  MoveL (T16343) to (117.45, 112.15, 17.7) mm, rotated rx 180 ry 0 rz -180 deg; joints [2.729, 71.249, -37.734, 4.933, -33.613, -4.112]
  Call Extruder 0.04881
  MoveL (T16344) to (118.18, 113.58, 17.7) mm, rotated rx 180 ry 0 rz -180 deg; joints [2.729, 71.249, -37.734, 4.933, -33.613, -4.112]
  Call Extruder 0.12804
  MoveL (T16345) to (121.16, 116.55, 17.7) mm, rotated rx 180 ry 0 rz -180 deg; joints [1.429, 67.441, -30.576, 2.381, -36.89, -1.905]
  Call Extruder 0.03385
  MoveL (T16346) to (121.16, 117.66, 17.7) mm, rotated rx 180 ry 0 rz -180 deg; joints [1.429, 67.441, -30.576, 2.381, -36.89, -1.905]
  Call Extruder 0.04175
  MoveL (T16347) to (120.19, 118.63, 17.7) mm, rotated rx 180 ry 0 rz -180 deg; joints [1.432, 67.145, -30.019, 2.372, -37.15, -1.891]
  Call Extruder 0.04741
  MoveL (T16348) to (120.19, 120.19, 17.7) mm, rotated rx 180 ry 0 rz -180 deg; joints [1.432, 67.145, -30.019, 2.372, -37.15, -1.891]
  Call Extruder 0.04175
  MoveL (T16349) to (121.16, 121.16, 17.7) mm, rotated rx 180 ry 0 rz -180 deg; joints [1.432, 67.145, -30.019, 2.372, -37.15, -1.891]
  Call Extruder 0.07441
  MoveL (T16350) to (121.16, 118.71, 17.7) mm, rotated rx 180 ry 0 rz -180 deg; joints [1.821, 66.26, -28.355, 2.962, -37.942, -2.336]
  Set speed (150.0 mm/s)
  MoveL (T16351) to (120.05, 117.4, 17.7) mm, rotated rx 180 ry 0 rz -180 deg; joints [1.821, 66.26, -28.355, 2.962, -37.942, -2.336]
  Set speed (50.0 mm/s)
  MoveL (T16352) to (120.05, 117.4, 17.7) mm, rotated rx 180 ry 0 rz -180 deg; joints [1.442, 66.234, -28.307, 2.345, -37.95, -1.849]
  Call Extruder 0.01089
  MoveL (T16353) to (119.96, 117.05, 17.7) mm, rotated rx 180 ry 0 rz -180 deg; joints [1.442, 66.234, -28.307, 2.345, -37.95, -1.849]
  Call Extruder 0.0635
  MoveL (T16354) to (119.01, 115.2, 17.7) mm, rotated rx 180 ry 0 rz -180 deg; joints [3.211, 71.325, -37.875, 5.812, -33.585, -4.847]
  Call Extruder 0.09231
  MoveL (T16355) to (121.16, 113.06, 17.7) mm, rotated rx 180 ry 0 rz -180 deg; joints [3.211, 71.325, -37.875, 5.812, -33.585, -4.847]
  Call Extruder 0.03385
  MoveL (T16356) to (121.16, 111.94, 17.7) mm, rotated rx 180 ry 0 rz -180 deg; joints [3.211, 71.325, -37.875, 5.812, -33.585, -4.847]
  Call Extruder 0.06789
  MoveL (T16357) to (119.58, 110.37, 17.7) mm, rotated rx 180 ry 0 rz -180 deg; joints [3.226, 70.568, -36.453, 5.738, -34.249, -4.748]
  Call Extruder 0.03053
  MoveL (T16358) to (120.29, 109.66, 17.7) mm, rotated rx 180 ry 0 rz -180 deg; joints [3.226, 70.568, -36.453, 5.738, -34.249, -4.748]
  Call Extruder 0.00661
  MoveL (T16359) to (120.37, 109.46, 17.7) mm, rotated rx 180 ry 0 rz -180 deg; joints [3.226, 70.568, -36.453, 5.738, -34.249, -4.748]
  Call Extruder 0.00686
  MoveL (T16360) to (120.37, 109.23, 17.7) mm, rotated rx 180 ry 0 rz -180 deg; joints [3.226, 70.568, -36.453, 5.738, -34.249, -4.748]
  Call Extruder 0.03378
  MoveL (T16361) to (121.16, 108.45, 17.7) mm, rotated rx 180 ry 0 rz -180 deg; joints [3.226, 70.568, -36.453, 5.738, -34.249, -4.748]
  Call Extruder 0.03385
  MoveL (T16362) to (121.16, 107.34, 17.7) mm, rotated rx 180 ry 0 rz -180 deg; joints [3.226, 70.568, -36.453, 5.738, -34.249, -4.748]
  Call Extruder 0.03378
  MoveL (T16363) to (120.37, 106.56, 17.7) mm, rotated rx 180 ry 0 rz -180 deg; joints [3.226, 70.568, -36.453, 5.738, -34.249, -4.748]
  Call Extruder 0.04531
  MoveL (T16364) to (120.37, 105.07, 17.7) mm, rotated rx 180 ry 0 rz -180 deg; joints [3.226, 70.568, -36.453, 5.738, -34.249, -4.748]
  Call Extruder 0.00661
  MoveL (T16365) to (120.29, 104.87, 17.7) mm, rotated rx 180 ry 0 rz -180 deg; joints [3.219, 70.895, -37.068, 5.77, -33.962, -4.79]
  Call Extruder 0.00334
  MoveL (T16366) to (120.21, 104.79, 17.7) mm, rotated rx 180 ry 0 rz -180 deg; joints [3.219, 70.895, -37.068, 5.77, -33.962, -4.79]
  Call Extruder 0.04071
  MoveL (T16367) to (121.16, 103.84, 17.7) mm, rotated rx 180 ry 0 rz -180 deg; joints [3.219, 70.895, -37.068, 5.77, -33.962, -4.79]
  Call Extruder 0.07441
  MoveL (T16368) to (121.16, 106.29, 17.7) mm, rotated rx 180 ry 0 rz -180 deg; joints [3.219, 70.895, -37.068, 5.77, -33.962, -4.79]
  Set speed (45.0 mm/s)
  Call Extruder -1.6
  MoveL (T16369) to (121.16, 106.29, 17.7) mm, rotated rx 180 ry 0 rz -180 deg; joints [3.219, 70.895, -37.068, 5.77, -33.962, -4.79]
  Set speed (120.0 mm/s)
  MoveL (T16370) to (121.16, 106.29, 17.7) mm, rotated rx 180 ry 0 rz -180 deg; joints [3.219, 70.895, -37.068, 5.77, -33.962, -4.79]
  Call Extruder -0.38
  MoveL (T16371) to (121.16, 105.22, 17.7) mm, rotated rx 180 ry 0 rz -180 deg; joints [3.219, 70.895, -37.068, 5.77, -33.962, -4.79]
  Set speed (45.0 mm/s)
  Call Extruder -0.02
  MoveL (T16372) to (121.16, 105.22, 17.7) mm, rotated rx 180 ry 0 rz -180 deg; joints [3.219, 70.895, -37.068, 5.77, -33.962, -4.79]
  Set speed (150.0 mm/s)
  MoveL (T16373) to (121.16, 105.22, 19.7) mm, rotated rx 180 ry 0 rz -180 deg; joints [1.407, 66.123, -28.505, 2.305, -37.64, -1.825]
  MoveL (T16374) to (120.15, 108.89, 19.7) mm, rotated rx 180 ry 0 rz -180 deg; joints [1.407, 66.336, -28.539, 2.296, -37.819, -1.814]
  MoveL (T16375) to (120.15, 108.89, 17.7) mm, rotated rx 180 ry 0 rz -180 deg; joints [1.407, 66.336, -28.539, 2.296, -37.819, -1.814]
  Set speed (40.0 mm/s)
  Call Extruder 2.0
  MoveL (T16376) to (120.15, 108.89, 17.7) mm, rotated rx 180 ry 0 rz -180 deg; joints [1.407, 66.336, -28.539, 2.296, -37.819, -1.814]
  Call Extruder 0.11511
  MoveL (T16377) to (117.48, 111.56, 17.7) mm, rotated rx 180 ry 0 rz -180 deg; joints [1.407, 66.336, -28.539, 2.296, -37.819, -1.814]
  Set speed (45.0 mm/s)
  Call Extruder -1.6
  MoveL (T16378) to (117.48, 111.56, 17.7) mm, rotated rx 180 ry 0 rz -180 deg; joints [1.407, 66.336, -28.539, 2.296, -37.819, -1.814]
  Set speed (120.0 mm/s)
  MoveL (T16379) to (117.48, 111.56, 17.7) mm, rotated rx 180 ry 0 rz -180 deg; joints [1.407, 66.336, -28.539, 2.296, -37.819, -1.814]
  Call Extruder -0.38
  MoveL (T16380) to (118.23, 110.8, 17.7) mm, rotated rx 180 ry 0 rz -180 deg; joints [1.407, 66.336, -28.539, 2.296, -37.819, -1.814]
  Set speed (45.0 mm/s)
  Call Extruder -0.02
  MoveL (T16381) to (118.23, 110.8, 17.7) mm, rotated rx 180 ry 0 rz -180 deg; joints [1.407, 66.336, -28.539, 2.296, -37.819, -1.814]
  Set speed (150.0 mm/s)
  MoveL (T16382) to (118.23, 110.8, 19.7) mm, rotated rx 180 ry 0 rz -180 deg; joints [1.407, 66.336, -28.539, 2.296, -37.819, -1.814]
  MoveL (T16383) to (118.65, 121.34, 19.7) mm, rotated rx 180 ry 0 rz -180 deg; joints [1.363, 71.176, -37.635, 2.466, -33.565, -2.055]
  MoveL (T16384) to (118.65, 121.34, 17.7) mm, rotated rx 180 ry 0 rz -180 deg; joints [1.363, 71.176, -37.635, 2.466, -33.565, -2.055]
  Set speed (40.0 mm/s)
  Call Extruder 2.0
  MoveL (T16385) to (118.65, 121.34, 17.7) mm, rotated rx 180 ry 0 rz -180 deg; joints [1.363, 71.176, -37.635, 2.466, -33.565, -2.055]
  Call Extruder 0.04796
  MoveL (T16386) to (119.76, 120.23, 17.7) mm, rotated rx 180 ry 0 rz -180 deg; joints [3.241, 71.403, -38.062, 5.883, -33.48, -4.912]
  Call Extruder 0.00166
  MoveL (T16387) to (119.78, 120.18, 17.7) mm, rotated rx 180 ry 0 rz -180 deg; joints [3.241, 71.403, -38.062, 5.883, -33.48, -4.912]
  Call Extruder 0.01669
  MoveL (T16388) to (119.78, 119.63, 17.7) mm, rotated rx 180 ry 0 rz -180 deg; joints [3.241, 71.403, -38.062, 5.883, -33.48, -4.912]
  Call Extruder 0.06581
  MoveL (T16389) to (118.25, 121.16, 17.7) mm, rotated rx 180 ry 0 rz -180 deg; joints [3.351, 66.321, -28.512, 5.456, -37.936, -4.308]
  Call Extruder 0.01758
  MoveL (T16390) to (117.68, 121.16, 17.7) mm, rotated rx 180 ry 0 rz -180 deg; joints [3.351, 66.321, -28.512, 5.456, -37.936, -4.308]
  Call Extruder 0.09068
  MoveL (T16391) to (119.78, 119.05, 17.7) mm, rotated rx 180 ry 0 rz -180 deg; joints [3.351, 66.321, -28.512, 5.456, -37.936, -4.308]
  Call Extruder 0.01758
  MoveL (T16392) to (119.78, 118.48, 17.7) mm, rotated rx 180 ry 0 rz -180 deg; joints [1.409, 66.13, -28.153, 2.29, -37.999, -1.805]
  Call Extruder 0.11554
  MoveL (T16393) to (117.1, 121.16, 17.7) mm, rotated rx 180 ry 0 rz -180 deg; joints [1.409, 66.13, -28.153, 2.29, -37.999, -1.805]
  Call Extruder 0.01758
  MoveL (T16394) to (116.52, 121.16, 17.7) mm, rotated rx 180 ry 0 rz -180 deg; joints [1.409, 66.13, -28.153, 2.29, -37.999, -1.805]
  Call Extruder 0.13957
  MoveL (T16395) to (119.76, 117.92, 17.7) mm, rotated rx 180 ry 0 rz -180 deg; joints [1.407, 66.32, -28.51, 2.295, -37.833, -1.813]
  Call Extruder 0.01457
  MoveL (T16396) to (119.65, 117.45, 17.7) mm, rotated rx 180 ry 0 rz -180 deg; joints [1.407, 66.32, -28.51, 2.295, -37.833, -1.813]
  Call Extruder 0.15961
  MoveL (T16397) to (115.95, 121.16, 17.7) mm, rotated rx 180 ry 0 rz -180 deg; joints [1.407, 66.32, -28.51, 2.295, -37.833, -1.813]
  Call Extruder 0.01758
  MoveL (T16398) to (115.37, 121.16, 17.7) mm, rotated rx 180 ry 0 rz -180 deg; joints [1.407, 66.32, -28.51, 2.295, -37.833, -1.813]
  Call Extruder 0.17783
  MoveL (T16399) to (119.49, 117.03, 17.7) mm, rotated rx 180 ry 0 rz -180 deg; joints [1.407, 66.32, -28.51, 2.295, -37.833, -1.813]
  Call Extruder 0.01306
  MoveL (T16400) to (119.3, 116.65, 17.7) mm, rotated rx 180 ry 0 rz -180 deg; joints [1.407, 66.32, -28.51, 2.295, -37.833, -1.813]
  Call Extruder 0.19428
  MoveL (T16401) to (114.8, 121.16, 17.7) mm, rotated rx 180 ry 0 rz -180 deg; joints [1.365, 66.126, -28.145, 2.218, -38.002, -1.748]
  Call Extruder 0.01758
  MoveL (T16402) to (114.22, 121.16, 17.7) mm, rotated rx 180 ry 0 rz -180 deg; joints [1.365, 66.126, -28.145, 2.218, -38.002, -1.748]
  Call Extruder 0.21073
  MoveL (T16403) to (119.1, 116.27, 17.7) mm, rotated rx 180 ry 0 rz -180 deg; joints [1.365, 66.126, -28.145, 2.218, -38.002, -1.748]
  Call Extruder 0.01306
  MoveL (T16404) to (118.91, 115.89, 17.7) mm, rotated rx 180 ry 0 rz -180 deg; joints [1.365, 66.126, -28.145, 2.218, -38.002, -1.748]
  Call Extruder 0.22717
  MoveL (T16405) to (113.64, 121.16, 17.7) mm, rotated rx 180 ry 0 rz -180 deg; joints [1.319, 71.301, -37.87, 2.394, -33.454, -1.998]
  Call Extruder 0.01758
  MoveL (T16406) to (113.07, 121.16, 17.7) mm, rotated rx 180 ry 0 rz -180 deg; joints [1.319, 71.301, -37.87, 2.394, -33.454, -1.998]
  Call Extruder 0.24362
  MoveL (T16407) to (118.71, 115.51, 17.7) mm, rotated rx 180 ry 0 rz -180 deg; joints [1.319, 71.301, -37.87, 2.394, -33.454, -1.998]
  Call Extruder 0.01306
  MoveL (T16408) to (118.52, 115.13, 17.7) mm, rotated rx 180 ry 0 rz -180 deg; joints [3.282, 71.54, -38.319, 5.974, -33.364, -4.995]
  Call Extruder 0.26007
  MoveL (T16409) to (112.49, 121.16, 17.7) mm, rotated rx 180 ry 0 rz -180 deg; joints [3.282, 71.54, -38.319, 5.974, -33.364, -4.995]
  Call Extruder 0.01758
  MoveL (T16410) to (111.91, 121.16, 17.7) mm, rotated rx 180 ry 0 rz -180 deg; joints [3.398, 66.223, -28.327, 5.521, -38.025, -4.354]
  Call Extruder 0.27651
  MoveL (T16411) to (118.32, 114.75, 17.7) mm, rotated rx 180 ry 0 rz -180 deg; joints [3.398, 66.223, -28.327, 5.521, -38.025, -4.354]
  Call Extruder 0.01306
  MoveL (T16412) to (118.13, 114.36, 17.7) mm, rotated rx 180 ry 0 rz -180 deg; joints [3.398, 66.223, -28.327, 5.521, -38.025, -4.354]
  Call Extruder 0.29296
  MoveL (T16413) to (111.34, 121.16, 17.7) mm, rotated rx 180 ry 0 rz -180 deg; joints [3.398, 66.223, -28.327, 5.521, -38.025, -4.354]
  Call Extruder 0.01758
  MoveL (T16414) to (110.76, 121.16, 17.7) mm, rotated rx 180 ry 0 rz -180 deg; joints [1.366, 66.024, -27.953, 2.215, -38.092, -1.744]
  Call Extruder 0.30941
  MoveL (T16415) to (117.93, 113.98, 17.7) mm, rotated rx 180 ry 0 rz -180 deg; joints [1.366, 66.024, -27.953, 2.215, -38.092, -1.744]
  Call Extruder 0.01306
  MoveL (T16416) to (117.74, 113.6, 17.7) mm, rotated rx 180 ry 0 rz -180 deg; joints [1.366, 66.024, -27.953, 2.215, -38.092, -1.744]
  Call Extruder 0.32585
  MoveL (T16417) to (110.18, 121.16, 17.7) mm, rotated rx 180 ry 0 rz -180 deg; joints [1.365, 66.111, -28.116, 2.217, -38.015, -1.747]
  Call Extruder 0.01758
  MoveL (T16418) to (109.61, 121.16, 17.7) mm, rotated rx 180 ry 0 rz -180 deg; joints [1.365, 66.111, -28.116, 2.217, -38.015, -1.747]
  Call Extruder 0.3423
  MoveL (T16419) to (117.54, 113.22, 17.7) mm, rotated rx 180 ry 0 rz -180 deg; joints [1.365, 66.111, -28.116, 2.217, -38.015, -1.747]
  Call Extruder 0.01306
  MoveL (T16420) to (117.35, 112.84, 17.7) mm, rotated rx 180 ry 0 rz -180 deg; joints [1.365, 66.111, -28.116, 2.217, -38.015, -1.747]
  Call Extruder 0.35875
  MoveL (T16421) to (109.03, 121.16, 17.7) mm, rotated rx 180 ry 0 rz -180 deg; joints [1.332, 65.919, -27.755, 2.156, -38.183, -1.695]
  Call Extruder 0.01758
  MoveL (T16422) to (108.45, 121.16, 17.7) mm, rotated rx 180 ry 0 rz -180 deg; joints [1.332, 65.919, -27.755, 2.156, -38.183, -1.695]
  Call Extruder 0.37519
  MoveL (T16423) to (117.15, 112.46, 17.7) mm, rotated rx 180 ry 0 rz -180 deg; joints [1.332, 65.919, -27.755, 2.156, -38.183, -1.695]
  Call Extruder 0.01306
  MoveL (T16424) to (116.96, 112.08, 17.7) mm, rotated rx 180 ry 0 rz -180 deg; joints [1.332, 65.919, -27.755, 2.156, -38.183, -1.695]
  Call Extruder 0.39164
  MoveL (T16425) to (107.88, 121.16, 17.7) mm, rotated rx 180 ry 0 rz -180 deg; joints [1.332, 65.919, -27.755, 2.156, -38.183, -1.695]
  Call Extruder 0.01758
  MoveL (T16426) to (107.3, 121.16, 17.7) mm, rotated rx 180 ry 0 rz -180 deg; joints [1.332, 65.919, -27.755, 2.156, -38.183, -1.695]
  Call Extruder 0.40809
  MoveL (T16427) to (116.76, 111.69, 17.7) mm, rotated rx 180 ry 0 rz -180 deg; joints [1.332, 65.919, -27.755, 2.156, -38.183, -1.695]
  Call Extruder 0.01107
  MoveL (T16428) to (116.6, 111.37, 17.7) mm, rotated rx 180 ry 0 rz -180 deg; joints [1.323, 65.918, -27.754, 2.141, -38.183, -1.683]
  Call Extruder 0.0149
  MoveL (T16429) to (117.09, 111.37, 17.7) mm, rotated rx 180 ry 0 rz -180 deg; joints [1.323, 65.918, -27.754, 2.141, -38.183, -1.683]
  Call Extruder 0.12417
  MoveL (T16430) to (119.96, 108.49, 17.7) mm, rotated rx 180 ry 0 rz -180 deg; joints [1.323, 65.918, -27.754, 2.141, -38.183, -1.683]
  Call Extruder 0.01758
  MoveL (T16431) to (119.96, 107.92, 17.7) mm, rotated rx 180 ry 0 rz -180 deg; joints [1.276, 71.427, -38.107, 2.322, -33.342, -1.94]
  Call Extruder 0.57106
  MoveL (T16432) to (106.73, 121.16, 17.7) mm, rotated rx 180 ry 0 rz -180 deg; joints [1.276, 71.427, -38.107, 2.322, -33.342, -1.94]
  Call Extruder 0.00679
  MoveL (T16433) to (106.5, 121.16, 17.7) mm, rotated rx 180 ry 0 rz -180 deg; joints [1.276, 71.427, -38.107, 2.322, -33.342, -1.94]
  Call Extruder 0.00763
  MoveL (T16434) to (106.33, 120.98, 17.7) mm, rotated rx 180 ry 0 rz -180 deg; joints [1.276, 71.427, -38.107, 2.322, -33.342, -1.94]
  Call Extruder 0.58829
  MoveL (T16435) to (119.96, 107.34, 17.7) mm, rotated rx 180 ry 0 rz -180 deg; joints [3.322, 71.677, -38.577, 6.066, -33.247, -5.079]
  Call Extruder 0.01758
  MoveL (T16436) to (119.96, 106.76, 17.7) mm, rotated rx 180 ry 0 rz -180 deg; joints [3.322, 71.677, -38.577, 6.066, -33.247, -5.079]
  Call Extruder 0.60072
  MoveL (T16437) to (106.04, 120.69, 17.7) mm, rotated rx 180 ry 0 rz -180 deg; joints [3.322, 71.677, -38.577, 6.066, -33.247, -5.079]
  Call Extruder 0.01243
  MoveL (T16438) to (105.75, 120.4, 17.7) mm, rotated rx 180 ry 0 rz -180 deg; joints [3.445, 66.125, -28.143, 5.586, -38.114, -4.4]
  Call Extruder 0.61315
  MoveL (T16439) to (119.96, 106.19, 17.7) mm, rotated rx 180 ry 0 rz -180 deg; joints [3.445, 66.125, -28.143, 5.586, -38.114, -4.4]
  Call Extruder 0.01758
  MoveL (T16440) to (119.96, 105.61, 17.7) mm, rotated rx 180 ry 0 rz -180 deg; joints [3.445, 66.125, -28.143, 5.586, -38.114, -4.4]
  Call Extruder 0.62159
  MoveL (T16441) to (105.55, 120.02, 17.7) mm, rotated rx 180 ry 0 rz -180 deg; joints [3.445, 66.125, -28.143, 5.586, -38.114, -4.4]
  Call Extruder 0.01758
  MoveL (T16442) to (105.55, 119.44, 17.7) mm, rotated rx 180 ry 0 rz -180 deg; joints [1.339, 65.919, -27.756, 2.166, -38.183, -1.703]
  Call Extruder 0.61978
  MoveL (T16443) to (119.92, 105.08, 17.7) mm, rotated rx 180 ry 0 rz -180 deg; joints [1.339, 65.919, -27.756, 2.166, -38.183, -1.703]
  Call Extruder 0.01243
  MoveL (T16444) to (119.63, 104.79, 17.7) mm, rotated rx 180 ry 0 rz -180 deg; joints [1.326, 65.933, -27.783, 2.146, -38.17, -1.687]
  Call Extruder 0.60735
  MoveL (T16445) to (105.55, 118.87, 17.7) mm, rotated rx 180 ry 0 rz -180 deg; joints [1.326, 65.933, -27.783, 2.146, -38.17, -1.687]
  Call Extruder 0.01758
  MoveL (T16446) to (105.55, 118.29, 17.7) mm, rotated rx 180 ry 0 rz -180 deg; joints [1.326, 65.933, -27.783, 2.146, -38.17, -1.687]
  Call Extruder 0.59492
  MoveL (T16447) to (119.35, 104.5, 17.7) mm, rotated rx 180 ry 0 rz -180 deg; joints [1.326, 65.933, -27.783, 2.146, -38.17, -1.687]
  Call Extruder 0.01243
  MoveL (T16448) to (119.06, 104.21, 17.7) mm, rotated rx 180 ry 0 rz -180 deg; joints [1.326, 65.933, -27.783, 2.146, -38.17, -1.687]
  Call Extruder 0.58249
  MoveL (T16449) to (105.55, 117.72, 17.7) mm, rotated rx 180 ry 0 rz -180 deg; joints [1.326, 65.933, -27.783, 2.146, -38.17, -1.687]
  Call Extruder 0.01758
  MoveL (T16450) to (105.55, 117.14, 17.7) mm, rotated rx 180 ry 0 rz -180 deg; joints [1.326, 65.933, -27.783, 2.146, -38.17, -1.687]
  Call Extruder 0.57006
  MoveL (T16451) to (118.77, 103.92, 17.7) mm, rotated rx 180 ry 0 rz -180 deg; joints [1.326, 65.933, -27.783, 2.146, -38.17, -1.687]
  Call Extruder 0.00343
  MoveL (T16452) to (118.69, 103.84, 17.7) mm, rotated rx 180 ry 0 rz -180 deg; joints [1.323, 65.918, -27.754, 2.141, -38.183, -1.683]
  Call Extruder 0.01274
  MoveL (T16453) to (118.27, 103.84, 17.7) mm, rotated rx 180 ry 0 rz -180 deg; joints [1.323, 65.918, -27.754, 2.141, -38.183, -1.683]
  Call Extruder 0.54862
  MoveL (T16454) to (105.55, 116.56, 17.7) mm, rotated rx 180 ry 0 rz -180 deg; joints [1.321, 66.153, -28.196, 2.147, -37.977, -1.693]
  Call Extruder 0.01758
  MoveL (T16455) to (105.55, 115.99, 17.7) mm, rotated rx 180 ry 0 rz -180 deg; joints [1.321, 66.153, -28.196, 2.147, -37.977, -1.693]
  Call Extruder 0.0956
  MoveL (T16456) to (107.77, 113.77, 17.7) mm, rotated rx 180 ry 0 rz -180 deg; joints [1.321, 66.153, -28.196, 2.147, -37.977, -1.693]
  Set speed (150.0 mm/s)
  MoveL (T16457) to (108.15, 113.39, 17.7) mm, rotated rx 180 ry 0 rz -180 deg; joints [1.321, 66.153, -28.196, 2.147, -37.977, -1.693]
  Set speed (40.0 mm/s)
  MoveL (T16458) to (108.15, 113.39, 17.7) mm, rotated rx 180 ry 0 rz -180 deg; joints [1.321, 66.153, -28.196, 2.147, -37.977, -1.693]
  Call Extruder 0.41176
  MoveL (T16459) to (117.7, 103.84, 17.7) mm, rotated rx 180 ry 0 rz -180 deg; joints [1.321, 66.153, -28.196, 2.147, -37.977, -1.693]
  Call Extruder 0.01758
  MoveL (T16460) to (117.12, 103.84, 17.7) mm, rotated rx 180 ry 0 rz -180 deg; joints [1.321, 66.153, -28.196, 2.147, -37.977, -1.693]
  Call Extruder 0.38942
  MoveL (T16461) to (108.09, 112.87, 17.7) mm, rotated rx 180 ry 0 rz -180 deg; joints [1.321, 66.153, -28.196, 2.147, -37.977, -1.693]
  Call Extruder 0.01307
  MoveL (T16462) to (107.9, 112.49, 17.7) mm, rotated rx 180 ry 0 rz -180 deg; joints [1.321, 65.916, -28.158, 2.157, -37.777, -1.705]
  Call Extruder 0.37296
  MoveL (T16463) to (116.54, 103.84, 17.7) mm, rotated rx 180 ry 0 rz -180 deg; joints [1.402, 70.099, -36.007, 2.501, -34.117, -2.071]
  Call Extruder 0.01758
  MoveL (T16464) to (115.97, 103.84, 17.7) mm, rotated rx 180 ry 0 rz -180 deg; joints [1.402, 70.099, -36.007, 2.501, -34.117, -2.071]
  Call Extruder 0.35649
  MoveL (T16465) to (107.7, 112.11, 17.7) mm, rotated rx 180 ry 0 rz -180 deg; joints [1.402, 70.332, -36.05, 2.488, -34.308, -2.056]
  Call Extruder 0.01307
  MoveL (T16466) to (107.51, 111.73, 17.7) mm, rotated rx 180 ry 0 rz -180 deg; joints [1.402, 70.332, -36.05, 2.488, -34.308, -2.056]
  Call Extruder 0.34003
  MoveL (T16467) to (115.39, 103.84, 17.7) mm, rotated rx 180 ry 0 rz -180 deg; joints [1.402, 70.332, -36.05, 2.488, -34.308, -2.056]
  Call Extruder 0.01758
  MoveL (T16468) to (114.81, 103.84, 17.7) mm, rotated rx 180 ry 0 rz -180 deg; joints [1.402, 70.332, -36.05, 2.488, -34.308, -2.056]
  Call Extruder 0.32357
  MoveL (T16469) to (107.31, 111.35, 17.7) mm, rotated rx 180 ry 0 rz -180 deg; joints [1.402, 70.332, -36.05, 2.488, -34.308, -2.056]
  Call Extruder 0.01307
  MoveL (T16470) to (107.12, 110.96, 17.7) mm, rotated rx 180 ry 0 rz -180 deg; joints [1.402, 70.332, -36.05, 2.488, -34.308, -2.056]
  Call Extruder 0.3071
  MoveL (T16471) to (114.24, 103.84, 17.7) mm, rotated rx 180 ry 0 rz -180 deg; joints [1.402, 70.332, -36.05, 2.488, -34.308, -2.056]
  Call Extruder 0.01758
  MoveL (T16472) to (113.66, 103.84, 17.7) mm, rotated rx 180 ry 0 rz -180 deg; joints [1.396, 71.083, -37.46, 2.52, -33.648, -2.098]
  Call Extruder 0.29064
  MoveL (T16473) to (106.92, 110.58, 17.7) mm, rotated rx 180 ry 0 rz -180 deg; joints [1.396, 71.083, -37.46, 2.52, -33.648, -2.098]
  Call Extruder 0.01307
  MoveL (T16474) to (106.73, 110.2, 17.7) mm, rotated rx 180 ry 0 rz -180 deg; joints [1.396, 71.083, -37.46, 2.52, -33.648, -2.098]
  Call Extruder 0.27417
  MoveL (T16475) to (113.08, 103.84, 17.7) mm, rotated rx 180 ry 0 rz -180 deg; joints [3.316, 66.395, -28.651, 5.407, -37.868, -4.274]
  Call Extruder 0.01758
  MoveL (T16476) to (112.51, 103.84, 17.7) mm, rotated rx 180 ry 0 rz -180 deg; joints [3.316, 66.395, -28.651, 5.407, -37.868, -4.274]
  Call Extruder 0.25771
  MoveL (T16477) to (106.53, 109.82, 17.7) mm, rotated rx 180 ry 0 rz -180 deg; joints [3.316, 66.395, -28.651, 5.407, -37.868, -4.274]
  Call Extruder 0.01307
  MoveL (T16478) to (106.34, 109.44, 17.7) mm, rotated rx 180 ry 0 rz -180 deg; joints [2.938, 66.346, -28.558, 4.788, -37.885, -3.782]
  Call Extruder 0.24124
  MoveL (T16479) to (111.93, 103.84, 17.7) mm, rotated rx 180 ry 0 rz -180 deg; joints [2.938, 66.346, -28.558, 4.788, -37.885, -3.782]
  Call Extruder 0.01758
  MoveL (T16480) to (111.36, 103.84, 17.7) mm, rotated rx 180 ry 0 rz -180 deg; joints [2.938, 66.346, -28.558, 4.788, -37.885, -3.782]
  Call Extruder 0.22478
  MoveL (T16481) to (106.14, 109.06, 17.7) mm, rotated rx 180 ry 0 rz -180 deg; joints [2.938, 66.346, -28.558, 4.788, -37.885, -3.782]
  Call Extruder 0.01307
  MoveL (T16482) to (105.95, 108.67, 17.7) mm, rotated rx 180 ry 0 rz -180 deg; joints [2.938, 66.346, -28.558, 4.788, -37.885, -3.782]
  Call Extruder 0.20831
  MoveL (T16483) to (110.78, 103.84, 17.7) mm, rotated rx 180 ry 0 rz -180 deg; joints [3.295, 67.312, -30.372, 5.471, -37.065, -4.371]
  Call Extruder 0.01758
  MoveL (T16484) to (110.2, 103.84, 17.7) mm, rotated rx 180 ry 0 rz -180 deg; joints [3.295, 67.312, -30.372, 5.471, -37.065, -4.371]
  Call Extruder 0.19185
  MoveL (T16485) to (105.75, 108.29, 17.7) mm, rotated rx 180 ry 0 rz -180 deg; joints [3.295, 67.312, -30.372, 5.471, -37.065, -4.371]
  Call Extruder 0.00693
  MoveL (T16486) to (105.65, 108.09, 17.7) mm, rotated rx 180 ry 0 rz -180 deg; joints [3.288, 67.61, -30.932, 5.493, -36.804, -4.403]
  Call Extruder 0.00686
  MoveL (T16487) to (105.6, 107.87, 17.7) mm, rotated rx 180 ry 0 rz -180 deg; joints [3.288, 67.61, -30.932, 5.493, -36.804, -4.403]
  Call Extruder 0.17364
  MoveL (T16488) to (109.63, 103.84, 17.7) mm, rotated rx 180 ry 0 rz -180 deg; joints [1.879, 71.124, -37.537, 3.395, -33.633, -2.827]
  Call Extruder 0.01758
  MoveL (T16489) to (109.05, 103.84, 17.7) mm, rotated rx 180 ry 0 rz -180 deg; joints [1.879, 71.124, -37.537, 3.395, -33.633, -2.827]
  Call Extruder 0.15359
  MoveL (T16490) to (105.49, 107.41, 17.7) mm, rotated rx 180 ry 0 rz -180 deg; joints [1.879, 71.124, -37.537, 3.395, -33.633, -2.827]
  Call Extruder 0.00278
  MoveL (T16491) to (105.47, 107.32, 17.7) mm, rotated rx 180 ry 0 rz -180 deg; joints [1.879, 71.124, -37.537, 3.395, -33.633, -2.827]
  Call Extruder 0.01427
  MoveL (T16492) to (105.47, 106.85, 17.7) mm, rotated rx 180 ry 0 rz -180 deg; joints [1.879, 71.124, -37.537, 3.395, -33.633, -2.827]
  Call Extruder 0.12957
  MoveL (T16493) to (108.47, 103.84, 17.7) mm, rotated rx 180 ry 0 rz -180 deg; joints [1.763, 71.113, -37.517, 3.183, -33.637, -2.651]
  Call Extruder 0.01758
  MoveL (T16494) to (107.9, 103.84, 17.7) mm, rotated rx 180 ry 0 rz -180 deg; joints [1.763, 71.113, -37.517, 3.183, -33.637, -2.651]
  Call Extruder 0.1047
  MoveL (T16495) to (105.47, 106.27, 17.7) mm, rotated rx 180 ry 0 rz -180 deg; joints [1.763, 71.113, -37.517, 3.183, -33.637, -2.651]
  Call Extruder 0.01758
  MoveL (T16496) to (105.47, 105.69, 17.7) mm, rotated rx 180 ry 0 rz -180 deg; joints [1.405, 70.017, -35.456, 2.476, -34.585, -2.039]
  Call Extruder 0.07984
  MoveL (T16497) to (107.32, 103.84, 17.7) mm, rotated rx 180 ry 0 rz -180 deg; joints [1.405, 70.017, -35.456, 2.476, -34.585, -2.039]
  Call Extruder 0.01758
  MoveL (T16498) to (106.75, 103.84, 17.7) mm, rotated rx 180 ry 0 rz -180 deg; joints [1.408, 69.688, -34.839, 2.463, -34.874, -2.021]
  Call Extruder 0.06288
  MoveL (T16499) to (105.29, 105.3, 17.7) mm, rotated rx 180 ry 0 rz -180 deg; joints [1.408, 69.688, -34.839, 2.463, -34.874, -2.021]
  Set speed (45.0 mm/s)
  Call Extruder -1.6
  MoveL (T16500) to (105.29, 105.3, 17.7) mm, rotated rx 180 ry 0 rz -180 deg; joints [2.818, 66.332, -28.531, 4.592, -37.89, -3.627]
  Set speed (120.0 mm/s)
  MoveL (T16501) to (105.29, 105.3, 17.7) mm, rotated rx 180 ry 0 rz -180 deg; joints [2.44, 66.29, -28.454, 3.973, -37.903, -3.137]
  Call Extruder -0.38
  MoveL (T16502) to (106.04, 104.55, 17.7) mm, rotated rx 180 ry 0 rz -180 deg; joints [2.44, 66.29, -28.454, 3.973, -37.903, -3.137]
  Set speed (45.0 mm/s)
  Call Extruder -0.02
  MoveL (T16503) to (106.04, 104.55, 17.7) mm, rotated rx 180 ry 0 rz -180 deg; joints [2.44, 66.29, -28.454, 3.973, -37.903, -3.137]
  Set speed (150.0 mm/s)
  MoveL (T16504) to (106.04, 104.55, 19.7) mm, rotated rx 180 ry 0 rz -180 deg; joints [3.266, 68.57, -32.736, 5.568, -35.962, -4.511]
  MoveL (T16505) to (104.34, 103.54, 19.7) mm, rotated rx 180 ry 0 rz -180 deg; joints [3.266, 68.57, -32.736, 5.568, -35.962, -4.511]
  MoveL (T16506) to (104.34, 103.54, 17.9) mm, rotated rx 180 ry 0 rz -180 deg; joints [3.266, 68.57, -32.736, 5.568, -35.962, -4.511]
  Set speed (40.0 mm/s)
  Call Extruder 2.0
  MoveL (T16507) to (104.34, 103.54, 17.9) mm, rotated rx 180 ry 0 rz -180 deg; joints [3.266, 68.57, -32.736, 5.568, -35.962, -4.511]
  Call Extruder 0.52159
  MoveL (T16508) to (121.46, 103.54, 17.9) mm, rotated rx 180 ry 0 rz -180 deg; joints [3.26, 68.883, -33.326, 5.593, -35.687, -4.548]
  Call Extruder 0.54596
  MoveL (T16509) to (121.46, 121.46, 17.9) mm, rotated rx 180 ry 0 rz -180 deg; joints [3.26, 68.883, -33.326, 5.593, -35.687, -4.548]
  Call Extruder 0.54596
  MoveL (T16510) to (103.54, 121.46, 17.9) mm, rotated rx 180 ry 0 rz -180 deg; joints [3.26, 68.883, -33.326, 5.593, -35.687, -4.548]
  Call Extruder 0.54596
  MoveL (T16511) to (103.54, 103.54, 17.9) mm, rotated rx 180 ry 0 rz -180 deg; joints [3.26, 68.883, -33.326, 5.593, -35.687, -4.548]
  Call Extruder 0.02254
  MoveL (T16512) to (104.28, 103.54, 17.9) mm, rotated rx 180 ry 0 rz -180 deg; joints [2.362, 71.177, -37.638, 4.27, -33.613, -3.558]
  Set speed (150.0 mm/s)
  MoveL (T16513) to (103.53, 103.13, 17.9) mm, rotated rx 180 ry 0 rz -180 deg; joints [2.362, 71.177, -37.638, 4.27, -33.613, -3.558]
  Set speed (40.0 mm/s)
  MoveL (T16514) to (103.53, 103.13, 17.9) mm, rotated rx 180 ry 0 rz -180 deg; joints [2.362, 71.177, -37.638, 4.27, -33.613, -3.558]
  Call Extruder 0.55858
  MoveL (T16515) to (121.87, 103.13, 17.9) mm, rotated rx 180 ry 0 rz -180 deg; joints [2.362, 71.177, -37.638, 4.27, -33.613, -3.558]
  Call Extruder 0.57077
  MoveL (T16516) to (121.87, 121.87, 17.9) mm, rotated rx 180 ry 0 rz -180 deg; joints [2.246, 71.163, -37.611, 4.059, -33.618, -3.382]
  Call Extruder 0.57077
  MoveL (T16517) to (103.13, 121.87, 17.9) mm, rotated rx 180 ry 0 rz -180 deg; joints [2.246, 71.163, -37.611, 4.059, -33.618, -3.382]
  Call Extruder 0.57077
  MoveL (T16518) to (103.13, 103.13, 17.9) mm, rotated rx 180 ry 0 rz -180 deg; joints [2.246, 71.163, -37.611, 4.059, -33.618, -3.382]
  Call Extruder 0.01036
  MoveL (T16519) to (103.47, 103.13, 17.9) mm, rotated rx 180 ry 0 rz -180 deg; joints [1.417, 68.683, -32.95, 2.425, -35.758, -1.969]
  Set speed (150.0 mm/s)
  MoveL (T16520) to (102.72, 102.81, 17.9) mm, rotated rx 180 ry 0 rz -180 deg; joints [1.417, 68.683, -32.95, 2.425, -35.758, -1.969]
  Set speed (25.0 mm/s)
  MoveL (T16521) to (102.72, 102.81, 17.9) mm, rotated rx 180 ry 0 rz -180 deg; joints [1.42, 68.372, -32.365, 2.414, -36.032, -1.953]
  Call Extruder 0.00259
  MoveL (T16522) to (102.72, 102.72, 17.9) mm, rotated rx 180 ry 0 rz -180 deg; joints [1.42, 68.372, -32.365, 2.414, -36.032, -1.953]
  Call Extruder 0.59557
  MoveL (T16523) to (122.28, 102.72, 17.9) mm, rotated rx 180 ry 0 rz -180 deg; joints [1.42, 68.372, -32.365, 2.414, -36.032, -1.953]
  Call Extruder 0.59557
  MoveL (T16524) to (122.28, 122.28, 17.9) mm, rotated rx 180 ry 0 rz -180 deg; joints [1.42, 68.372, -32.365, 2.414, -36.032, -1.953]
  Call Extruder 0.59557
  MoveL (T16525) to (102.72, 122.28, 17.9) mm, rotated rx 180 ry 0 rz -180 deg; joints [2.319, 66.279, -28.432, 3.777, -37.907, -2.982]
  Call Extruder 0.59115
  MoveL (T16526) to (102.72, 102.87, 17.9) mm, rotated rx 180 ry 0 rz -180 deg; joints [2.319, 66.279, -28.432, 3.777, -37.907, -2.982]
  Set speed (150.0 mm/s)
  MoveL (T16527) to (102.78, 102.75, 17.9) mm, rotated rx 180 ry 0 rz -180 deg; joints [1.941, 66.245, -28.369, 3.159, -37.919, -2.493]
  Set speed (45.0 mm/s)
  Call Extruder -1.6
  MoveL (T16528) to (102.78, 102.75, 17.9) mm, rotated rx 180 ry 0 rz -180 deg; joints [1.941, 66.245, -28.369, 3.159, -37.919, -2.493]
  Set speed (120.0 mm/s)
  MoveL (T16529) to (102.78, 102.75, 17.9) mm, rotated rx 180 ry 0 rz -180 deg; joints [3.239, 69.895, -35.228, 5.681, -34.799, -4.67]
  Call Extruder -0.05166
  MoveL (T16530) to (102.72, 102.72, 17.9) mm, rotated rx 180 ry 0 rz -180 deg; joints [3.239, 69.895, -35.228, 5.681, -34.799, -4.67]
  Call Extruder -0.32834
  MoveL (T16531) to (103.65, 102.72, 17.9) mm, rotated rx 180 ry 0 rz -180 deg; joints [3.239, 69.895, -35.228, 5.681, -34.799, -4.67]
  Set speed (45.0 mm/s)
  Call Extruder -0.02
  MoveL (T16532) to (103.65, 102.72, 17.9) mm, rotated rx 180 ry 0 rz -180 deg; joints [3.232, 70.227, -35.851, 5.711, -34.509, -4.711]
  Set speed (150.0 mm/s)
  MoveL (T16533) to (103.65, 102.72, 19.9) mm, rotated rx 180 ry 0 rz -180 deg; joints [2.845, 71.243, -37.761, 5.148, -33.588, -4.292]
  MoveL (T16534) to (106.08, 103.93, 19.9) mm, rotated rx 180 ry 0 rz -180 deg; joints [2.845, 71.243, -37.761, 5.148, -33.588, -4.292]
  MoveL (T16535) to (106.08, 103.93, 17.9) mm, rotated rx 180 ry 0 rz -180 deg; joints [2.845, 71.243, -37.761, 5.148, -33.588, -4.292]
  Set speed (40.0 mm/s)
  Call Extruder 2.0
  MoveL (T16536) to (106.08, 103.93, 17.9) mm, rotated rx 180 ry 0 rz -180 deg; joints [2.845, 71.243, -37.761, 5.148, -33.588, -4.292]
  Set speed (50.0 mm/s)
  MoveL (T16537) to (106.08, 103.93, 17.9) mm, rotated rx 180 ry 0 rz -180 deg; joints [2.729, 71.226, -37.729, 4.936, -33.595, -4.115]
  Call Extruder 0.00361
  MoveL (T16538) to (106.17, 103.84, 17.9) mm, rotated rx 180 ry 0 rz -180 deg; joints [2.729, 71.226, -37.729, 4.936, -33.595, -4.115]
  Call Extruder 0.0708
  MoveL (T16539) to (103.84, 103.84, 17.9) mm, rotated rx 180 ry 0 rz -180 deg; joints [2.729, 71.226, -37.729, 4.936, -33.595, -4.115]
  Call Extruder 0.05255
  MoveL (T16540) to (105.06, 105.06, 17.9) mm, rotated rx 180 ry 0 rz -180 deg; joints [2.729, 71.226, -37.729, 4.936, -33.595, -4.115]
  Call Extruder 0.03217
  MoveL (T16541) to (105.06, 106.12, 17.9) mm, rotated rx 180 ry 0 rz -180 deg; joints [1.429, 67.418, -30.572, 2.382, -36.87, -1.906]
  Call Extruder 0.0525
  MoveL (T16542) to (103.84, 107.34, 17.9) mm, rotated rx 180 ry 0 rz -180 deg; joints [1.429, 67.418, -30.572, 2.382, -36.87, -1.906]
  Call Extruder 0.03385
  MoveL (T16543) to (103.84, 108.45, 17.9) mm, rotated rx 180 ry 0 rz -180 deg; joints [1.432, 67.122, -30.015, 2.373, -37.13, -1.892]
  Call Extruder 0.13495
  MoveL (T16544) to (106.98, 111.58, 17.9) mm, rotated rx 180 ry 0 rz -180 deg; joints [1.432, 67.122, -30.015, 2.373, -37.13, -1.892]
  Call Extruder 0.04156
  MoveL (T16545) to (107.6, 112.8, 17.9) mm, rotated rx 180 ry 0 rz -180 deg; joints [1.432, 67.122, -30.015, 2.373, -37.13, -1.892]
  Call Extruder 0.16166
  MoveL (T16546) to (103.84, 116.55, 17.9) mm, rotated rx 180 ry 0 rz -180 deg; joints [1.821, 66.236, -28.351, 2.963, -37.922, -2.338]
  Call Extruder 0.03385
  MoveL (T16547) to (103.84, 117.66, 17.9) mm, rotated rx 180 ry 0 rz -180 deg; joints [1.821, 66.236, -28.351, 2.963, -37.922, -2.338]
  Call Extruder 0.05612
  MoveL (T16548) to (105.15, 118.96, 17.9) mm, rotated rx 180 ry 0 rz -180 deg; joints [1.821, 66.236, -28.351, 2.963, -37.922, -2.338]
  Call Extruder 0.02709
  MoveL (T16549) to (105.15, 119.85, 17.9) mm, rotated rx 180 ry 0 rz -180 deg; joints [1.821, 66.236, -28.351, 2.963, -37.922, -2.338]
  Call Extruder 0.05612
  MoveL (T16550) to (103.84, 121.16, 17.9) mm, rotated rx 180 ry 0 rz -180 deg; joints [1.442, 66.21, -28.303, 2.346, -37.93, -1.851]
  Call Extruder 0.06345
  MoveL (T16551) to (105.93, 121.16, 17.9) mm, rotated rx 180 ry 0 rz -180 deg; joints [1.442, 66.21, -28.303, 2.346, -37.93, -1.851]
  Call Extruder 0.01096
  MoveL (T16552) to (105.67, 120.9, 17.9) mm, rotated rx 180 ry 0 rz -180 deg; joints [1.442, 66.21, -28.303, 2.346, -37.93, -1.851]
  Set speed (45.0 mm/s)
  Call Extruder -1.6
  MoveL (T16553) to (105.67, 120.9, 17.9) mm, rotated rx 180 ry 0 rz -180 deg; joints [3.211, 71.301, -37.871, 5.815, -33.566, -4.85]
  Set speed (120.0 mm/s)
  MoveL (T16554) to (105.67, 120.9, 17.9) mm, rotated rx 180 ry 0 rz -180 deg; joints [3.211, 71.301, -37.871, 5.815, -33.566, -4.85]
  Call Extruder -0.12811
  MoveL (T16555) to (105.93, 121.16, 17.9) mm, rotated rx 180 ry 0 rz -180 deg; joints [3.226, 70.545, -36.448, 5.741, -34.23, -4.752]
  Call Extruder -0.25189
  MoveL (T16556) to (105.22, 121.16, 17.9) mm, rotated rx 180 ry 0 rz -180 deg; joints [3.226, 70.545, -36.448, 5.741, -34.23, -4.752]
  Set speed (45.0 mm/s)
  Call Extruder -0.02
  MoveL (T16557) to (105.22, 121.16, 17.9) mm, rotated rx 180 ry 0 rz -180 deg; joints [3.226, 70.545, -36.448, 5.741, -34.23, -4.752]
  Set speed (150.0 mm/s)
  MoveL (T16558) to (105.22, 121.16, 19.9) mm, rotated rx 180 ry 0 rz -180 deg; joints [3.226, 70.545, -36.448, 5.741, -34.23, -4.752]
  MoveL (T16559) to (105.15, 117.23, 19.9) mm, rotated rx 180 ry 0 rz -180 deg; joints [3.226, 70.545, -36.448, 5.741, -34.23, -4.752]
  MoveL (T16560) to (105.15, 117.23, 17.9) mm, rotated rx 180 ry 0 rz -180 deg; joints [3.226, 70.545, -36.448, 5.741, -34.23, -4.752]
  Set speed (40.0 mm/s)
  Call Extruder 2.0
  MoveL (T16561) to (105.15, 117.23, 17.9) mm, rotated rx 180 ry 0 rz -180 deg; joints [3.226, 70.545, -36.448, 5.741, -34.23, -4.752]
  Set speed (50.0 mm/s)
  MoveL (T16562) to (105.15, 117.23, 17.9) mm, rotated rx 180 ry 0 rz -180 deg; joints [3.226, 70.545, -36.448, 5.741, -34.23, -4.752]
  Call Extruder 0.04143
  MoveL (T16563) to (105.15, 115.87, 17.9) mm, rotated rx 180 ry 0 rz -180 deg; joints [3.226, 70.545, -36.448, 5.741, -34.23, -4.752]
  Call Extruder 0.00661
  MoveL (T16564) to (105.23, 115.67, 17.9) mm, rotated rx 180 ry 0 rz -180 deg; joints [3.219, 70.872, -37.064, 5.772, -33.943, -4.794]
  Call Extruder 0.02637
  MoveL (T16565) to (105.84, 115.05, 17.9) mm, rotated rx 180 ry 0 rz -180 deg; joints [3.219, 70.872, -37.064, 5.772, -33.943, -4.794]
  Call Extruder 0.08606
  MoveL (T16566) to (103.84, 113.06, 17.9) mm, rotated rx 180 ry 0 rz -180 deg; joints [3.219, 70.872, -37.064, 5.772, -33.943, -4.794]
  Call Extruder 0.03385
  MoveL (T16567) to (103.84, 111.94, 17.9) mm, rotated rx 180 ry 0 rz -180 deg; joints [3.219, 70.872, -37.064, 5.772, -33.943, -4.794]
  Call Extruder 0.09463
  MoveL (T16568) to (106.04, 109.75, 17.9) mm, rotated rx 180 ry 0 rz -180 deg; joints [3.219, 70.872, -37.064, 5.772, -33.943, -4.794]
  Call Extruder 0.05062
  MoveL (T16569) to (105.29, 108.27, 17.9) mm, rotated rx 180 ry 0 rz -180 deg; joints [3.219, 70.872, -37.064, 5.772, -33.943, -4.794]
  Call Extruder 0.02377
  MoveL (T16570) to (105.1, 107.51, 17.9) mm, rotated rx 180 ry 0 rz -180 deg; joints [3.219, 70.872, -37.064, 5.772, -33.943, -4.794]
  Set speed (45.0 mm/s)
  Call Extruder -1.6
  MoveL (T16571) to (105.1, 107.51, 17.9) mm, rotated rx 180 ry 0 rz -180 deg; joints [3.219, 70.638, -37.02, 5.801, -33.754, -4.828]
  Set speed (120.0 mm/s)
  MoveL (T16572) to (105.1, 107.51, 17.9) mm, rotated rx 180 ry 0 rz -180 deg; joints [1.407, 66.099, -28.501, 2.306, -37.62, -1.827]
  Call Extruder -0.278
  MoveL (T16573) to (105.29, 108.27, 17.9) mm, rotated rx 180 ry 0 rz -180 deg; joints [1.407, 66.312, -28.535, 2.297, -37.799, -1.815]
  Call Extruder -0.102
  MoveL (T16574) to (105.42, 108.52, 17.9) mm, rotated rx 180 ry 0 rz -180 deg; joints [1.407, 66.312, -28.535, 2.297, -37.799, -1.815]
  Set speed (45.0 mm/s)
  Call Extruder -0.02
  MoveL (T16575) to (105.42, 108.52, 17.9) mm, rotated rx 180 ry 0 rz -180 deg; joints [1.407, 66.312, -28.535, 2.297, -37.799, -1.815]
  Set speed (150.0 mm/s)
  MoveL (T16576) to (105.42, 108.52, 19.9) mm, rotated rx 180 ry 0 rz -180 deg; joints [1.407, 66.312, -28.535, 2.297, -37.799, -1.815]
  MoveL (T16577) to (118.51, 103.66, 19.9) mm, rotated rx 180 ry 0 rz -180 deg; joints [1.407, 66.312, -28.535, 2.297, -37.799, -1.815]
  MoveL (T16578) to (118.51, 103.66, 17.9) mm, rotated rx 180 ry 0 rz -180 deg; joints [1.407, 66.312, -28.535, 2.297, -37.799, -1.815]
  Set speed (40.0 mm/s)
  Call Extruder 2.0
  MoveL (T16579) to (118.51, 103.66, 17.9) mm, rotated rx 180 ry 0 rz -180 deg; joints [1.407, 66.312, -28.535, 2.297, -37.799, -1.815]
  Call Extruder 0.06226
  MoveL (T16580) to (119.94, 105.1, 17.9) mm, rotated rx 180 ry 0 rz -180 deg; joints [1.407, 66.312, -28.535, 2.297, -37.799, -1.815]
  Call Extruder 0.00161
  MoveL (T16581) to (119.96, 105.15, 17.9) mm, rotated rx 180 ry 0 rz -180 deg; joints [1.407, 66.312, -28.535, 2.297, -37.799, -1.815]
  Call Extruder 0.01683
  MoveL (T16582) to (119.96, 105.7, 17.9) mm, rotated rx 180 ry 0 rz -180 deg; joints [1.363, 71.152, -37.63, 2.467, -33.546, -2.057]
  Call Extruder 0.08024
  MoveL (T16583) to (118.11, 103.84, 17.9) mm, rotated rx 180 ry 0 rz -180 deg; joints [1.363, 71.152, -37.63, 2.467, -33.546, -2.057]
  Call Extruder 0.0177
  MoveL (T16584) to (117.53, 103.84, 17.9) mm, rotated rx 180 ry 0 rz -180 deg; joints [1.363, 71.152, -37.63, 2.467, -33.546, -2.057]
  Call Extruder 0.10527
  MoveL (T16585) to (119.96, 106.28, 17.9) mm, rotated rx 180 ry 0 rz -180 deg; joints [1.363, 71.152, -37.63, 2.467, -33.546, -2.057]
  Call Extruder 0.0177
  MoveL (T16586) to (119.96, 106.86, 17.9) mm, rotated rx 180 ry 0 rz -180 deg; joints [1.363, 71.152, -37.63, 2.467, -33.546, -2.057]
  Call Extruder 0.1303
  MoveL (T16587) to (116.95, 103.84, 17.9) mm, rotated rx 180 ry 0 rz -180 deg; joints [3.241, 71.379, -38.057, 5.886, -33.461, -4.916]
  Call Extruder 0.0177
  MoveL (T16588) to (116.38, 103.84, 17.9) mm, rotated rx 180 ry 0 rz -180 deg; joints [3.241, 71.379, -38.057, 5.886, -33.461, -4.916]
  Call Extruder 0.15533
  MoveL (T16589) to (119.96, 107.43, 17.9) mm, rotated rx 180 ry 0 rz -180 deg; joints [3.241, 71.379, -38.057, 5.886, -33.461, -4.916]
  Call Extruder 0.0177
  MoveL (T16590) to (119.96, 108.01, 17.9) mm, rotated rx 180 ry 0 rz -180 deg; joints [3.351, 66.298, -28.508, 5.459, -37.916, -4.311]
  Call Extruder 0.18036
  MoveL (T16591) to (115.8, 103.84, 17.9) mm, rotated rx 180 ry 0 rz -180 deg; joints [3.351, 66.298, -28.508, 5.459, -37.916, -4.311]
  Call Extruder 0.0177
  MoveL (T16592) to (115.22, 103.84, 17.9) mm, rotated rx 180 ry 0 rz -180 deg; joints [3.351, 66.298, -28.508, 5.459, -37.916, -4.311]
  Call Extruder 0.20539
  MoveL (T16593) to (119.96, 108.59, 17.9) mm, rotated rx 180 ry 0 rz -180 deg; joints [1.409, 66.107, -28.149, 2.291, -37.98, -1.806]
  Call Extruder 0.0177
  MoveL (T16594) to (119.96, 109.17, 17.9) mm, rotated rx 180 ry 0 rz -180 deg; joints [1.409, 66.107, -28.149, 2.291, -37.98, -1.806]
  Call Extruder 0.23042
  MoveL (T16595) to (114.64, 103.84, 17.9) mm, rotated rx 180 ry 0 rz -180 deg; joints [1.409, 66.107, -28.149, 2.291, -37.98, -1.806]
  Call Extruder 0.0177
  MoveL (T16596) to (114.06, 103.84, 17.9) mm, rotated rx 180 ry 0 rz -180 deg; joints [1.409, 66.107, -28.149, 2.291, -37.98, -1.806]
  Call Extruder 0.24813
  MoveL (T16597) to (119.8, 109.58, 17.9) mm, rotated rx 180 ry 0 rz -180 deg; joints [1.407, 66.296, -28.506, 2.296, -37.813, -1.814]
  Call Extruder 0.01252
  MoveL (T16598) to (119.51, 109.87, 17.9) mm, rotated rx 180 ry 0 rz -180 deg; joints [1.407, 66.296, -28.506, 2.296, -37.813, -1.814]
  Call Extruder 0.26064
  MoveL (T16599) to (113.48, 103.84, 17.9) mm, rotated rx 180 ry 0 rz -180 deg; joints [1.365, 66.102, -28.141, 2.219, -37.982, -1.749]
  Call Extruder 0.0177
  MoveL (T16600) to (112.91, 103.84, 17.9) mm, rotated rx 180 ry 0 rz -180 deg; joints [1.365, 66.102, -28.141, 2.219, -37.982, -1.749]
  Call Extruder 0.27316
  MoveL (T16601) to (119.22, 110.16, 17.9) mm, rotated rx 180 ry 0 rz -180 deg; joints [1.365, 66.102, -28.141, 2.219, -37.982, -1.749]
  Call Extruder 0.01252
  MoveL (T16602) to (118.93, 110.44, 17.9) mm, rotated rx 180 ry 0 rz -180 deg; joints [1.365, 66.102, -28.141, 2.219, -37.982, -1.749]
  Call Extruder 0.28567
  MoveL (T16603) to (112.33, 103.84, 17.9) mm, rotated rx 180 ry 0 rz -180 deg; joints [1.365, 66.102, -28.141, 2.219, -37.982, -1.749]
  Call Extruder 0.0177
  MoveL (T16604) to (111.75, 103.84, 17.9) mm, rotated rx 180 ry 0 rz -180 deg; joints [1.365, 66.102, -28.141, 2.219, -37.982, -1.749]
  Call Extruder 0.29819
  MoveL (T16605) to (118.64, 110.73, 17.9) mm, rotated rx 180 ry 0 rz -180 deg; joints [1.319, 71.277, -37.865, 2.395, -33.435, -1.999]
  Call Extruder 0.01252
  MoveL (T16606) to (118.35, 111.02, 17.9) mm, rotated rx 180 ry 0 rz -180 deg; joints [1.319, 71.277, -37.865, 2.395, -33.435, -1.999]
  Call Extruder 0.3107
  MoveL (T16607) to (111.17, 103.84, 17.9) mm, rotated rx 180 ry 0 rz -180 deg; joints [1.319, 71.277, -37.865, 2.395, -33.435, -1.999]
  Call Extruder 0.0177
  MoveL (T16608) to (110.59, 103.84, 17.9) mm, rotated rx 180 ry 0 rz -180 deg; joints [3.282, 71.516, -38.314, 5.977, -33.345, -4.999]
  Call Extruder 0.32322
  MoveL (T16609) to (118.06, 111.31, 17.9) mm, rotated rx 180 ry 0 rz -180 deg; joints [3.282, 71.516, -38.314, 5.977, -33.345, -4.999]
  Call Extruder 0.00328
  MoveL (T16610) to (117.97, 111.37, 17.9) mm, rotated rx 180 ry 0 rz -180 deg; joints [3.398, 66.199, -28.323, 5.524, -38.005, -4.357]
  Call Extruder 0.01316
  MoveL (T16611) to (117.54, 111.37, 17.9) mm, rotated rx 180 ry 0 rz -180 deg; joints [3.398, 66.199, -28.323, 5.524, -38.005, -4.357]
  Call Extruder 0.32579
  MoveL (T16612) to (110.01, 103.84, 17.9) mm, rotated rx 180 ry 0 rz -180 deg; joints [3.398, 66.199, -28.323, 5.524, -38.005, -4.357]
  Call Extruder 0.0177
  MoveL (T16613) to (109.44, 103.84, 17.9) mm, rotated rx 180 ry 0 rz -180 deg; joints [1.366, 66, -27.949, 2.216, -38.072, -1.745]
  Call Extruder 0.32579
  MoveL (T16614) to (116.96, 111.37, 17.9) mm, rotated rx 180 ry 0 rz -180 deg; joints [1.366, 66, -27.949, 2.216, -38.072, -1.745]
  Call Extruder 0.01118
  MoveL (T16615) to (116.6, 111.37, 17.9) mm, rotated rx 180 ry 0 rz -180 deg; joints [1.365, 66.087, -28.112, 2.218, -37.995, -1.749]
  Call Extruder 0.015
  MoveL (T16616) to (116.82, 111.81, 17.9) mm, rotated rx 180 ry 0 rz -180 deg; joints [1.365, 66.087, -28.112, 2.218, -37.995, -1.749]
  Call Extruder 0.34467
  MoveL (T16617) to (108.86, 103.84, 17.9) mm, rotated rx 180 ry 0 rz -180 deg; joints [1.365, 66.087, -28.112, 2.218, -37.995, -1.749]
  Call Extruder 0.0177
  MoveL (T16618) to (108.28, 103.84, 17.9) mm, rotated rx 180 ry 0 rz -180 deg; joints [1.332, 65.895, -27.751, 2.157, -38.163, -1.696]
  Call Extruder 0.39594
  MoveL (T16619) to (117.43, 112.99, 17.9) mm, rotated rx 180 ry 0 rz -180 deg; joints [1.332, 65.895, -27.751, 2.157, -38.163, -1.696]
  Call Extruder 0.04072
  MoveL (T16620) to (118.03, 114.18, 17.9) mm, rotated rx 180 ry 0 rz -180 deg; joints [1.332, 65.895, -27.751, 2.157, -38.163, -1.696]
  Call Extruder 0.4472
  MoveL (T16621) to (107.7, 103.84, 17.9) mm, rotated rx 180 ry 0 rz -180 deg; joints [1.332, 65.895, -27.751, 2.157, -38.163, -1.696]
  Call Extruder 0.0177
  MoveL (T16622) to (107.12, 103.84, 17.9) mm, rotated rx 180 ry 0 rz -180 deg; joints [1.332, 65.895, -27.751, 2.157, -38.163, -1.696]
  Call Extruder 0.49847
  MoveL (T16623) to (118.64, 115.36, 17.9) mm, rotated rx 180 ry 0 rz -180 deg; joints [1.332, 65.895, -27.751, 2.157, -38.163, -1.696]
  Call Extruder 0.04072
  MoveL (T16624) to (119.25, 116.55, 17.9) mm, rotated rx 180 ry 0 rz -180 deg; joints [1.332, 65.895, -27.751, 2.157, -38.163, -1.696]
  Call Extruder 0.54539
  MoveL (T16625) to (106.64, 103.94, 17.9) mm, rotated rx 180 ry 0 rz -180 deg; joints [1.323, 65.894, -27.75, 2.142, -38.163, -1.684]
  Call Extruder 0.01252
  MoveL (T16626) to (106.36, 104.23, 17.9) mm, rotated rx 180 ry 0 rz -180 deg; joints [1.276, 71.403, -38.102, 2.323, -33.323, -1.941]
  Call Extruder 0.57634
  MoveL (T16627) to (119.67, 117.55, 17.9) mm, rotated rx 180 ry 0 rz -180 deg; joints [1.276, 71.403, -38.102, 2.323, -33.323, -1.941]
  Call Extruder 0.01389
  MoveL (T16628) to (119.78, 117.99, 17.9) mm, rotated rx 180 ry 0 rz -180 deg; joints [1.276, 71.403, -38.102, 2.323, -33.323, -1.941]
  Call Extruder 0.00751
  MoveL (T16629) to (119.78, 118.24, 17.9) mm, rotated rx 180 ry 0 rz -180 deg; joints [1.276, 71.403, -38.102, 2.323, -33.323, -1.941]
  Call Extruder 0.59354
  MoveL (T16630) to (106.07, 104.52, 17.9) mm, rotated rx 180 ry 0 rz -180 deg; joints [1.276, 71.403, -38.102, 2.323, -33.323, -1.941]
  Call Extruder 0.01252
  MoveL (T16631) to (105.78, 104.81, 17.9) mm, rotated rx 180 ry 0 rz -180 deg; joints [3.322, 71.654, -38.573, 6.069, -33.228, -5.083]
  Call Extruder 0.60606
  MoveL (T16632) to (119.78, 118.81, 17.9) mm, rotated rx 180 ry 0 rz -180 deg; joints [3.322, 71.654, -38.573, 6.069, -33.228, -5.083]
  Call Extruder 0.0177
  MoveL (T16633) to (119.78, 119.39, 17.9) mm, rotated rx 180 ry 0 rz -180 deg; joints [3.322, 71.654, -38.573, 6.069, -33.228, -5.083]
  Call Extruder 0.6185
  MoveL (T16634) to (105.49, 105.1, 17.9) mm, rotated rx 180 ry 0 rz -180 deg; joints [3.445, 66.101, -28.14, 5.589, -38.094, -4.403]
  Call Extruder 0.0015
  MoveL (T16635) to (105.47, 105.15, 17.9) mm, rotated rx 180 ry 0 rz -180 deg; joints [3.445, 66.101, -28.14, 5.589, -38.094, -4.403]
  Call Extruder 0.01574
  MoveL (T16636) to (105.47, 105.66, 17.9) mm, rotated rx 180 ry 0 rz -180 deg; joints [3.445, 66.101, -28.14, 5.589, -38.094, -4.403]
  Call Extruder 0.61932
  MoveL (T16637) to (119.78, 119.97, 17.9) mm, rotated rx 180 ry 0 rz -180 deg; joints [1.339, 65.895, -27.752, 2.167, -38.163, -1.704]
  Call Extruder 0.00627
  MoveL (T16638) to (119.78, 120.18, 17.9) mm, rotated rx 180 ry 0 rz -180 deg; joints [1.339, 65.895, -27.752, 2.167, -38.163, -1.704]
  Call Extruder 0.00169
  MoveL (T16639) to (119.76, 120.23, 17.9) mm, rotated rx 180 ry 0 rz -180 deg; joints [1.339, 65.895, -27.752, 2.167, -38.163, -1.704]
  Call Extruder 0.00653
  MoveL (T16640) to (119.61, 120.38, 17.9) mm, rotated rx 180 ry 0 rz -180 deg; joints [1.339, 65.895, -27.752, 2.167, -38.163, -1.704]
  Call Extruder 0.61188
  MoveL (T16641) to (105.47, 106.24, 17.9) mm, rotated rx 180 ry 0 rz -180 deg; joints [1.326, 65.91, -27.779, 2.147, -38.15, -1.688]
  Call Extruder 0.0177
  MoveL (T16642) to (105.47, 106.82, 17.9) mm, rotated rx 180 ry 0 rz -180 deg; joints [1.326, 65.91, -27.779, 2.147, -38.15, -1.688]
  Call Extruder 0.59936
  MoveL (T16643) to (119.32, 120.67, 17.9) mm, rotated rx 180 ry 0 rz -180 deg; joints [1.326, 65.91, -27.779, 2.147, -38.15, -1.688]
  Call Extruder 0.01252
  MoveL (T16644) to (119.03, 120.96, 17.9) mm, rotated rx 180 ry 0 rz -180 deg; joints [1.326, 65.91, -27.779, 2.147, -38.15, -1.688]
  Call Extruder 0.58584
  MoveL (T16645) to (105.49, 107.42, 17.9) mm, rotated rx 180 ry 0 rz -180 deg; joints [1.326, 65.91, -27.779, 2.147, -38.15, -1.688]
  Call Extruder 0.02102
  MoveL (T16646) to (105.65, 108.09, 17.9) mm, rotated rx 180 ry 0 rz -180 deg; joints [1.326, 65.91, -27.779, 2.147, -38.15, -1.688]
  Call Extruder 0.0048
  MoveL (T16647) to (105.72, 108.23, 17.9) mm, rotated rx 180 ry 0 rz -180 deg; joints [1.326, 65.91, -27.779, 2.147, -38.15, -1.688]
  Call Extruder 0.55945
  MoveL (T16648) to (118.65, 121.16, 17.9) mm, rotated rx 180 ry 0 rz -180 deg; joints [1.323, 65.894, -27.75, 2.142, -38.163, -1.684]
  Call Extruder 0.0177
  MoveL (T16649) to (118.07, 121.16, 17.9) mm, rotated rx 180 ry 0 rz -180 deg; joints [1.323, 65.894, -27.75, 2.142, -38.163, -1.684]
  Call Extruder 0.50836
  MoveL (T16650) to (106.33, 109.41, 17.9) mm, rotated rx 180 ry 0 rz -180 deg; joints [1.321, 66.129, -28.192, 2.148, -37.957, -1.694]
  Call Extruder 0.04056
  MoveL (T16651) to (106.93, 110.59, 17.9) mm, rotated rx 180 ry 0 rz -180 deg; joints [1.321, 66.129, -28.192, 2.148, -37.957, -1.694]
  Call Extruder 0.45726
  MoveL (T16652) to (117.49, 121.16, 17.9) mm, rotated rx 180 ry 0 rz -180 deg; joints [1.321, 66.129, -28.192, 2.148, -37.957, -1.694]
  Call Extruder 0.0177
  MoveL (T16653) to (116.92, 121.16, 17.9) mm, rotated rx 180 ry 0 rz -180 deg; joints [1.321, 66.129, -28.192, 2.148, -37.957, -1.694]
  Call Extruder 0.40616
  MoveL (T16654) to (107.53, 111.77, 17.9) mm, rotated rx 180 ry 0 rz -180 deg; joints [1.321, 66.129, -28.192, 2.148, -37.957, -1.694]
  Call Extruder 0.04056
  MoveL (T16655) to (108.13, 112.95, 17.9) mm, rotated rx 180 ry 0 rz -180 deg; joints [1.321, 66.129, -28.192, 2.148, -37.957, -1.694]
  Call Extruder 0.35507
  MoveL (T16656) to (116.34, 121.16, 17.9) mm, rotated rx 180 ry 0 rz -180 deg; joints [1.321, 66.129, -28.192, 2.148, -37.957, -1.694]
  Call Extruder 0.0177
  MoveL (T16657) to (115.76, 121.16, 17.9) mm, rotated rx 180 ry 0 rz -180 deg; joints [1.321, 66.129, -28.192, 2.148, -37.957, -1.694]
  Call Extruder 0.31171
  MoveL (T16658) to (108.56, 113.95, 17.9) mm, rotated rx 180 ry 0 rz -180 deg; joints [1.402, 70.076, -36.003, 2.502, -34.098, -2.072]
  Call Extruder 0.0177
  MoveL (T16659) to (107.98, 113.95, 17.9) mm, rotated rx 180 ry 0 rz -180 deg; joints [1.402, 70.309, -36.045, 2.49, -34.289, -2.057]
  Call Extruder 0.31171
  MoveL (T16660) to (115.18, 121.16, 17.9) mm, rotated rx 180 ry 0 rz -180 deg; joints [1.402, 70.309, -36.045, 2.49, -34.289, -2.057]
  Call Extruder 0.0177
  MoveL (T16661) to (114.6, 121.16, 17.9) mm, rotated rx 180 ry 0 rz -180 deg; joints [1.402, 70.309, -36.045, 2.49, -34.289, -2.057]
  Call Extruder 0.30914
  MoveL (T16662) to (107.46, 114.01, 17.9) mm, rotated rx 180 ry 0 rz -180 deg; joints [1.402, 70.309, -36.045, 2.49, -34.289, -2.057]
  Call Extruder 0.01252
  MoveL (T16663) to (107.17, 114.3, 17.9) mm, rotated rx 180 ry 0 rz -180 deg; joints [1.402, 70.309, -36.045, 2.49, -34.289, -2.057]
  Call Extruder 0.29663
  MoveL (T16664) to (114.02, 121.16, 17.9) mm, rotated rx 180 ry 0 rz -180 deg; joints [1.402, 70.309, -36.045, 2.49, -34.289, -2.057]
  Call Extruder 0.0177
  MoveL (T16665) to (113.44, 121.16, 17.9) mm, rotated rx 180 ry 0 rz -180 deg; joints [1.402, 70.309, -36.045, 2.49, -34.289, -2.057]
  Call Extruder 0.28411
  MoveL (T16666) to (106.88, 114.59, 17.9) mm, rotated rx 180 ry 0 rz -180 deg; joints [1.402, 70.309, -36.045, 2.49, -34.289, -2.057]
  Call Extruder 0.01252
  MoveL (T16667) to (106.59, 114.88, 17.9) mm, rotated rx 180 ry 0 rz -180 deg; joints [1.402, 70.309, -36.045, 2.49, -34.289, -2.057]
  Call Extruder 0.2716
  MoveL (T16668) to (112.87, 121.16, 17.9) mm, rotated rx 180 ry 0 rz -180 deg; joints [1.402, 70.309, -36.045, 2.49, -34.289, -2.057]
  Call Extruder 0.0177
  MoveL (T16669) to (112.29, 121.16, 17.9) mm, rotated rx 180 ry 0 rz -180 deg; joints [1.402, 70.309, -36.045, 2.49, -34.289, -2.057]
  Call Extruder 0.25908
  MoveL (T16670) to (106.3, 115.17, 17.9) mm, rotated rx 180 ry 0 rz -180 deg; joints [1.396, 71.059, -37.455, 2.521, -33.629, -2.1]
  Call Extruder 0.01252
  MoveL (T16671) to (106.01, 115.46, 17.9) mm, rotated rx 180 ry 0 rz -180 deg; joints [1.396, 71.059, -37.455, 2.521, -33.629, -2.1]
  Call Extruder 0.24657
  MoveL (T16672) to (111.71, 121.16, 17.9) mm, rotated rx 180 ry 0 rz -180 deg; joints [1.396, 71.059, -37.455, 2.521, -33.629, -2.1]
  Call Extruder 0.0177
  MoveL (T16673) to (111.13, 121.16, 17.9) mm, rotated rx 180 ry 0 rz -180 deg; joints [1.396, 71.059, -37.455, 2.521, -33.629, -2.1]
  Call Extruder 0.23405
  MoveL (T16674) to (105.72, 115.75, 17.9) mm, rotated rx 180 ry 0 rz -180 deg; joints [3.316, 66.372, -28.647, 5.41, -37.849, -4.277]
  Call Extruder 0.00641
  MoveL (T16675) to (105.58, 115.9, 17.9) mm, rotated rx 180 ry 0 rz -180 deg; joints [3.316, 66.372, -28.647, 5.41, -37.849, -4.277]
  Call Extruder 0.00169
  MoveL (T16676) to (105.55, 115.95, 17.9) mm, rotated rx 180 ry 0 rz -180 deg; joints [3.316, 66.372, -28.647, 5.41, -37.849, -4.277]
  Call Extruder 0.00643
  MoveL (T16677) to (105.55, 116.16, 17.9) mm, rotated rx 180 ry 0 rz -180 deg; joints [3.316, 66.372, -28.647, 5.41, -37.849, -4.277]
  Call Extruder 0.21634
  MoveL (T16678) to (110.55, 121.16, 17.9) mm, rotated rx 180 ry 0 rz -180 deg; joints [3.316, 66.372, -28.647, 5.41, -37.849, -4.277]
  Call Extruder 0.0177
  MoveL (T16679) to (109.97, 121.16, 17.9) mm, rotated rx 180 ry 0 rz -180 deg; joints [2.938, 66.322, -28.554, 4.79, -37.865, -3.785]
  Call Extruder 0.19131
  MoveL (T16680) to (105.55, 116.73, 17.9) mm, rotated rx 180 ry 0 rz -180 deg; joints [2.938, 66.322, -28.554, 4.79, -37.865, -3.785]
  Call Extruder 0.0177
  MoveL (T16681) to (105.55, 117.31, 17.9) mm, rotated rx 180 ry 0 rz -180 deg; joints [3.295, 67.288, -30.368, 5.474, -37.046, -4.374]
  Call Extruder 0.16628
  MoveL (T16682) to (109.4, 121.16, 17.9) mm, rotated rx 180 ry 0 rz -180 deg; joints [3.295, 67.288, -30.368, 5.474, -37.046, -4.374]
  Call Extruder 0.0177
  MoveL (T16683) to (108.82, 121.16, 17.9) mm, rotated rx 180 ry 0 rz -180 deg; joints [3.295, 67.288, -30.368, 5.474, -37.046, -4.374]
  Call Extruder 0.14125
  MoveL (T16684) to (105.55, 117.89, 17.9) mm, rotated rx 180 ry 0 rz -180 deg; joints [3.295, 67.288, -30.368, 5.474, -37.046, -4.374]
  Call Extruder 0.0177
  MoveL (T16685) to (105.55, 118.47, 17.9) mm, rotated rx 180 ry 0 rz -180 deg; joints [3.288, 67.586, -30.928, 5.496, -36.785, -4.406]
  Call Extruder 0.11622
  MoveL (T16686) to (108.24, 121.16, 17.9) mm, rotated rx 180 ry 0 rz -180 deg; joints [3.288, 67.586, -30.928, 5.496, -36.785, -4.406]
  Call Extruder 0.0177
  MoveL (T16687) to (107.66, 121.16, 17.9) mm, rotated rx 180 ry 0 rz -180 deg; joints [3.288, 67.586, -30.928, 5.496, -36.785, -4.406]
  Call Extruder 0.09119
  MoveL (T16688) to (105.55, 119.05, 17.9) mm, rotated rx 180 ry 0 rz -180 deg; joints [1.879, 71.1, -37.533, 3.396, -33.614, -2.829]
  Call Extruder 0.0177
  MoveL (T16689) to (105.55, 119.63, 17.9) mm, rotated rx 180 ry 0 rz -180 deg; joints [1.879, 71.1, -37.533, 3.396, -33.614, -2.829]
  Call Extruder 0.06616
  MoveL (T16690) to (107.08, 121.16, 17.9) mm, rotated rx 180 ry 0 rz -180 deg; joints [1.763, 71.089, -37.512, 3.185, -33.618, -2.653]
  Call Extruder 0.0177
  MoveL (T16691) to (106.5, 121.16, 17.9) mm, rotated rx 180 ry 0 rz -180 deg; joints [1.763, 71.089, -37.512, 3.185, -33.618, -2.653]
  Call Extruder 0.04905
  MoveL (T16692) to (105.37, 120.02, 17.9) mm, rotated rx 180 ry 0 rz -180 deg; joints [1.405, 69.993, -35.452, 2.477, -34.566, -2.04]
  Set speed (45.0 mm/s)
  Call Extruder -1.6
  MoveL (T16693) to (105.37, 120.02, 17.9) mm, rotated rx 180 ry 0 rz -180 deg; joints [1.405, 69.993, -35.452, 2.477, -34.566, -2.04]
  Set speed (120.0 mm/s)
  MoveL (T16694) to (105.37, 120.02, 17.9) mm, rotated rx 180 ry 0 rz -180 deg; joints [1.405, 69.993, -35.452, 2.477, -34.566, -2.04]
  Call Extruder -0.38
  MoveL (T16695) to (106.12, 120.78, 17.9) mm, rotated rx 180 ry 0 rz -180 deg; joints [1.405, 69.993, -35.452, 2.477, -34.566, -2.04]
  Set speed (45.0 mm/s)
  Call Extruder -0.02
  MoveL (T16696) to (106.12, 120.78, 17.9) mm, rotated rx 180 ry 0 rz -180 deg; joints [1.408, 69.665, -34.834, 2.464, -34.855, -2.022]
  Set speed (150.0 mm/s)
  MoveL (T16697) to (106.12, 120.78, 19.9) mm, rotated rx 180 ry 0 rz -180 deg; joints [1.408, 69.665, -34.834, 2.464, -34.855, -2.022]
  MoveL (T16698) to (120.05, 117.4, 19.9) mm, rotated rx 180 ry 0 rz -180 deg; joints [1.408, 69.665, -34.834, 2.464, -34.855, -2.022]
  MoveL (T16699) to (120.05, 117.4, 17.9) mm, rotated rx 180 ry 0 rz -180 deg; joints [2.818, 66.308, -28.527, 4.594, -37.87, -3.629]
  Set speed (40.0 mm/s)
  Call Extruder 2.0
  MoveL (T16700) to (120.05, 117.4, 17.9) mm, rotated rx 180 ry 0 rz -180 deg; joints [2.818, 66.308, -28.527, 4.594, -37.87, -3.629]
  Set speed (50.0 mm/s)
  MoveL (T16701) to (120.05, 117.4, 17.9) mm, rotated rx 180 ry 0 rz -180 deg; joints [2.818, 66.308, -28.527, 4.594, -37.87, -3.629]
  Call Extruder 0.01089
  MoveL (T16702) to (119.96, 117.05, 17.9) mm, rotated rx 180 ry 0 rz -180 deg; joints [2.44, 66.267, -28.45, 3.975, -37.884, -3.139]
  Call Extruder 0.0635
  MoveL (T16703) to (119.01, 115.2, 17.9) mm, rotated rx 180 ry 0 rz -180 deg; joints [2.44, 66.267, -28.45, 3.975, -37.884, -3.139]
  Call Extruder 0.09231
  MoveL (T16704) to (121.16, 113.06, 17.9) mm, rotated rx 180 ry 0 rz -180 deg; joints [2.44, 66.267, -28.45, 3.975, -37.884, -3.139]
  Call Extruder 0.03385
  MoveL (T16705) to (121.16, 111.94, 17.9) mm, rotated rx 180 ry 0 rz -180 deg; joints [2.44, 66.267, -28.45, 3.975, -37.884, -3.139]
  Call Extruder 0.06789
  MoveL (T16706) to (119.58, 110.37, 17.9) mm, rotated rx 180 ry 0 rz -180 deg; joints [3.266, 68.546, -32.732, 5.57, -35.943, -4.515]
  Call Extruder 0.03053
  MoveL (T16707) to (120.29, 109.66, 17.9) mm, rotated rx 180 ry 0 rz -180 deg; joints [3.266, 68.546, -32.732, 5.57, -35.943, -4.515]
  Call Extruder 0.00661
  MoveL (T16708) to (120.37, 109.46, 17.9) mm, rotated rx 180 ry 0 rz -180 deg; joints [3.266, 68.546, -32.732, 5.57, -35.943, -4.515]
  Call Extruder 0.00686
  MoveL (T16709) to (120.37, 109.23, 17.9) mm, rotated rx 180 ry 0 rz -180 deg; joints [3.266, 68.546, -32.732, 5.57, -35.943, -4.515]
  Call Extruder 0.03378
  MoveL (T16710) to (121.16, 108.45, 17.9) mm, rotated rx 180 ry 0 rz -180 deg; joints [3.266, 68.546, -32.732, 5.57, -35.943, -4.515]
  Call Extruder 0.03385
  MoveL (T16711) to (121.16, 107.34, 17.9) mm, rotated rx 180 ry 0 rz -180 deg; joints [3.26, 68.86, -33.321, 5.596, -35.668, -4.551]
  Call Extruder 0.03378
  MoveL (T16712) to (120.37, 106.56, 17.9) mm, rotated rx 180 ry 0 rz -180 deg; joints [3.26, 68.86, -33.321, 5.596, -35.668, -4.551]
  Call Extruder 0.04531
  MoveL (T16713) to (120.37, 105.07, 17.9) mm, rotated rx 180 ry 0 rz -180 deg; joints [3.26, 68.86, -33.321, 5.596, -35.668, -4.551]
  Call Extruder 0.00661
  MoveL (T16714) to (120.29, 104.87, 17.9) mm, rotated rx 180 ry 0 rz -180 deg; joints [3.26, 68.86, -33.321, 5.596, -35.668, -4.551]
  Call Extruder 0.00334
  MoveL (T16715) to (120.21, 104.79, 17.9) mm, rotated rx 180 ry 0 rz -180 deg; joints [2.362, 71.154, -37.633, 4.272, -33.594, -3.561]
  Call Extruder 0.04071
  MoveL (T16716) to (121.16, 103.84, 17.9) mm, rotated rx 180 ry 0 rz -180 deg; joints [2.362, 71.154, -37.633, 4.272, -33.594, -3.561]
  Call Extruder 0.07441
  MoveL (T16717) to (121.16, 106.29, 17.9) mm, rotated rx 180 ry 0 rz -180 deg; joints [2.362, 71.154, -37.633, 4.272, -33.594, -3.561]
  Set speed (45.0 mm/s)
  Call Extruder -1.6
  MoveL (T16718) to (121.16, 106.29, 17.9) mm, rotated rx 180 ry 0 rz -180 deg; joints [2.246, 71.14, -37.607, 4.061, -33.599, -3.384]
  Set speed (120.0 mm/s)
  MoveL (T16719) to (121.16, 106.29, 17.9) mm, rotated rx 180 ry 0 rz -180 deg; joints [2.246, 71.14, -37.607, 4.061, -33.599, -3.384]
  Call Extruder -0.38
  MoveL (T16720) to (121.16, 105.22, 17.9) mm, rotated rx 180 ry 0 rz -180 deg; joints [1.417, 68.66, -32.946, 2.426, -35.739, -1.97]
  Set speed (45.0 mm/s)
  Call Extruder -0.02
  MoveL (T16721) to (121.16, 105.22, 17.9) mm, rotated rx 180 ry 0 rz -180 deg; joints [1.417, 68.66, -32.946, 2.426, -35.739, -1.97]
  Set speed (150.0 mm/s)
  MoveL (T16722) to (121.16, 105.22, 19.9) mm, rotated rx 180 ry 0 rz -180 deg; joints [1.42, 68.348, -32.361, 2.415, -36.012, -1.954]
  MoveL (T16723) to (119.44, 110.51, 19.9) mm, rotated rx 180 ry 0 rz -180 deg; joints [1.42, 68.348, -32.361, 2.415, -36.012, -1.954]
  MoveL (T16724) to (119.44, 110.51, 17.9) mm, rotated rx 180 ry 0 rz -180 deg; joints [2.319, 66.255, -28.428, 3.779, -37.888, -2.984]
  Set speed (40.0 mm/s)
  Call Extruder 2.0
  MoveL (T16725) to (119.44, 110.51, 17.9) mm, rotated rx 180 ry 0 rz -180 deg; joints [2.319, 66.255, -28.428, 3.779, -37.888, -2.984]
  Set speed (50.0 mm/s)
  MoveL (T16726) to (119.44, 110.51, 17.9) mm, rotated rx 180 ry 0 rz -180 deg; joints [2.319, 66.255, -28.428, 3.779, -37.888, -2.984]
  Call Extruder 0.05098
  MoveL (T16727) to (118.25, 111.7, 17.9) mm, rotated rx 180 ry 0 rz -180 deg; joints [2.319, 66.255, -28.428, 3.779, -37.888, -2.984]
  Call Extruder 0.00661
  MoveL (T16728) to (118.05, 111.78, 17.9) mm, rotated rx 180 ry 0 rz -180 deg; joints [1.941, 66.221, -28.365, 3.161, -37.899, -2.495]
  Call Extruder 0.00686
  MoveL (T16729) to (117.83, 111.78, 17.9) mm, rotated rx 180 ry 0 rz -180 deg; joints [1.941, 66.221, -28.365, 3.161, -37.899, -2.495]
  Call Extruder 0.01607
  MoveL (T16730) to (117.45, 112.15, 17.9) mm, rotated rx 180 ry 0 rz -180 deg; joints [1.941, 66.221, -28.365, 3.161, -37.899, -2.495]
  Call Extruder 0.04881
  MoveL (T16731) to (118.18, 113.58, 17.9) mm, rotated rx 180 ry 0 rz -180 deg; joints [3.239, 69.872, -35.224, 5.684, -34.78, -4.673]
  Call Extruder 0.12804
  MoveL (T16732) to (121.16, 116.55, 17.9) mm, rotated rx 180 ry 0 rz -180 deg; joints [3.239, 69.872, -35.224, 5.684, -34.78, -4.673]
  Call Extruder 0.03385
  MoveL (T16733) to (121.16, 117.66, 17.9) mm, rotated rx 180 ry 0 rz -180 deg; joints [3.239, 69.872, -35.224, 5.684, -34.78, -4.673]
  Call Extruder 0.04175
  MoveL (T16734) to (120.19, 118.63, 17.9) mm, rotated rx 180 ry 0 rz -180 deg; joints [3.239, 69.872, -35.224, 5.684, -34.78, -4.673]
  Call Extruder 0.04741
  MoveL (T16735) to (120.19, 120.19, 17.9) mm, rotated rx 180 ry 0 rz -180 deg; joints [3.232, 70.203, -35.846, 5.714, -34.49, -4.715]
  Call Extruder 0.04175
  MoveL (T16736) to (121.16, 121.16, 17.9) mm, rotated rx 180 ry 0 rz -180 deg; joints [3.232, 70.203, -35.846, 5.714, -34.49, -4.715]
  Call Extruder 0.07441
  MoveL (T16737) to (121.16, 118.71, 17.9) mm, rotated rx 180 ry 0 rz -180 deg; joints [3.232, 70.203, -35.846, 5.714, -34.49, -4.715]
  Set speed (45.0 mm/s)
  Call Extruder -1.6
  MoveL (T16738) to (121.16, 118.71, 17.9) mm, rotated rx 180 ry 0 rz -180 deg; joints [3.232, 70.203, -35.846, 5.714, -34.49, -4.715]
  Set speed (120.0 mm/s)
  MoveL (T16739) to (121.16, 118.71, 17.9) mm, rotated rx 180 ry 0 rz -180 deg; joints [2.845, 71.22, -37.757, 5.15, -33.57, -4.295]
  Call Extruder -0.38
  MoveL (T16740) to (121.16, 119.78, 17.9) mm, rotated rx 180 ry 0 rz -180 deg; joints [2.845, 71.22, -37.757, 5.15, -33.57, -4.295]
  Set speed (45.0 mm/s)
  Call Extruder -0.02
  MoveL (T16741) to (121.16, 119.78, 17.9) mm, rotated rx 180 ry 0 rz -180 deg; joints [2.845, 71.22, -37.757, 5.15, -33.57, -4.295]
  Set speed (150.0 mm/s)
  MoveL (T16742) to (121.16, 119.78, 19.9) mm, rotated rx 180 ry 0 rz -180 deg; joints [2.845, 71.22, -37.757, 5.15, -33.57, -4.295]
  MoveL (T16743) to (104.34, 103.54, 19.9) mm, rotated rx 180 ry 0 rz -180 deg; joints [2.729, 71.203, -37.725, 4.938, -33.576, -4.117]
  MoveL (T16744) to (104.34, 103.54, 18.1) mm, rotated rx 180 ry 0 rz -180 deg; joints [2.729, 71.203, -37.725, 4.938, -33.576, -4.117]
  Set speed (40.0 mm/s)
  Call Extruder 2.0
  MoveL (T16745) to (104.34, 103.54, 18.1) mm, rotated rx 180 ry 0 rz -180 deg; joints [2.729, 71.203, -37.725, 4.938, -33.576, -4.117]
  Call Extruder 0.52159
  MoveL (T16746) to (121.46, 103.54, 18.1) mm, rotated rx 180 ry 0 rz -180 deg; joints [1.429, 67.394, -30.568, 2.384, -36.85, -1.908]
  Call Extruder 0.54596
  MoveL (T16747) to (121.46, 121.46, 18.1) mm, rotated rx 180 ry 0 rz -180 deg; joints [1.429, 67.394, -30.568, 2.384, -36.85, -1.908]
  Call Extruder 0.54596
  MoveL (T16748) to (103.54, 121.46, 18.1) mm, rotated rx 180 ry 0 rz -180 deg; joints [1.432, 67.098, -30.011, 2.374, -37.11, -1.894]
  Call Extruder 0.54596
  MoveL (T16749) to (103.54, 103.54, 18.1) mm, rotated rx 180 ry 0 rz -180 deg; joints [1.432, 67.098, -30.011, 2.374, -37.11, -1.894]
  Call Extruder 0.02254
  MoveL (T16750) to (104.28, 103.54, 18.1) mm, rotated rx 180 ry 0 rz -180 deg; joints [1.432, 67.098, -30.011, 2.374, -37.11, -1.894]
  Set speed (150.0 mm/s)
  MoveL (T16751) to (103.53, 103.13, 18.1) mm, rotated rx 180 ry 0 rz -180 deg; joints [1.432, 67.098, -30.011, 2.374, -37.11, -1.894]
  Set speed (40.0 mm/s)
  MoveL (T16752) to (103.53, 103.13, 18.1) mm, rotated rx 180 ry 0 rz -180 deg; joints [1.821, 66.212, -28.347, 2.964, -37.902, -2.34]
  Call Extruder 0.55858
  MoveL (T16753) to (121.87, 103.13, 18.1) mm, rotated rx 180 ry 0 rz -180 deg; joints [1.821, 66.212, -28.347, 2.964, -37.902, -2.34]
  Call Extruder 0.57077
  MoveL (T16754) to (121.87, 121.87, 18.1) mm, rotated rx 180 ry 0 rz -180 deg; joints [1.821, 66.212, -28.347, 2.964, -37.902, -2.34]
  Call Extruder 0.57077
  MoveL (T16755) to (103.13, 121.87, 18.1) mm, rotated rx 180 ry 0 rz -180 deg; joints [1.442, 66.187, -28.299, 2.347, -37.91, -1.852]
  Call Extruder 0.57077
  MoveL (T16756) to (103.13, 103.13, 18.1) mm, rotated rx 180 ry 0 rz -180 deg; joints [1.442, 66.187, -28.299, 2.347, -37.91, -1.852]
  Call Extruder 0.01036
  MoveL (T16757) to (103.47, 103.13, 18.1) mm, rotated rx 180 ry 0 rz -180 deg; joints [1.442, 66.187, -28.299, 2.347, -37.91, -1.852]
  Set speed (150.0 mm/s)
  MoveL (T16758) to (102.72, 102.81, 18.1) mm, rotated rx 180 ry 0 rz -180 deg; joints [1.442, 66.187, -28.299, 2.347, -37.91, -1.852]
  Set speed (25.0 mm/s)
  MoveL (T16759) to (102.72, 102.81, 18.1) mm, rotated rx 180 ry 0 rz -180 deg; joints [3.211, 71.278, -37.866, 5.818, -33.548, -4.854]
  Call Extruder 0.00259
  MoveL (T16760) to (102.72, 102.72, 18.1) mm, rotated rx 180 ry 0 rz -180 deg; joints [3.226, 70.521, -36.444, 5.744, -34.211, -4.755]
  Call Extruder 0.59557
  MoveL (T16761) to (122.28, 102.72, 18.1) mm, rotated rx 180 ry 0 rz -180 deg; joints [3.226, 70.521, -36.444, 5.744, -34.211, -4.755]
  Call Extruder 0.59557
  MoveL (T16762) to (122.28, 122.28, 18.1) mm, rotated rx 180 ry 0 rz -180 deg; joints [3.226, 70.521, -36.444, 5.744, -34.211, -4.755]
  Call Extruder 0.59557
  MoveL (T16763) to (102.72, 122.28, 18.1) mm, rotated rx 180 ry 0 rz -180 deg; joints [3.226, 70.521, -36.444, 5.744, -34.211, -4.755]
  Call Extruder 0.59115
  MoveL (T16764) to (102.72, 102.87, 18.1) mm, rotated rx 180 ry 0 rz -180 deg; joints [3.226, 70.521, -36.444, 5.744, -34.211, -4.755]
  Set speed (150.0 mm/s)
  MoveL (T16765) to (102.78, 102.75, 18.1) mm, rotated rx 180 ry 0 rz -180 deg; joints [3.226, 70.521, -36.444, 5.744, -34.211, -4.755]
  Set speed (45.0 mm/s)
  Call Extruder -1.6
  MoveL (T16766) to (102.78, 102.75, 18.1) mm, rotated rx 180 ry 0 rz -180 deg; joints [3.226, 70.521, -36.444, 5.744, -34.211, -4.755]
  Set speed (120.0 mm/s)
  MoveL (T16767) to (102.78, 102.75, 18.1) mm, rotated rx 180 ry 0 rz -180 deg; joints [3.226, 70.521, -36.444, 5.744, -34.211, -4.755]
  Call Extruder -0.05166
  MoveL (T16768) to (102.72, 102.72, 18.1) mm, rotated rx 180 ry 0 rz -180 deg; joints [3.226, 70.521, -36.444, 5.744, -34.211, -4.755]
  Call Extruder -0.32834
  MoveL (T16769) to (103.65, 102.72, 18.1) mm, rotated rx 180 ry 0 rz -180 deg; joints [3.226, 70.521, -36.444, 5.744, -34.211, -4.755]
  Set speed (45.0 mm/s)
  Call Extruder -0.02
  MoveL (T16770) to (103.65, 102.72, 18.1) mm, rotated rx 180 ry 0 rz -180 deg; joints [3.226, 70.521, -36.444, 5.744, -34.211, -4.755]
  Set speed (150.0 mm/s)
  MoveL (T16771) to (103.65, 102.72, 20.1) mm, rotated rx 180 ry 0 rz -180 deg; joints [3.219, 70.848, -37.059, 5.775, -33.924, -4.797]
  MoveL (T16772) to (106.29, 103.84, 20.1) mm, rotated rx 180 ry 0 rz -180 deg; joints [3.219, 70.848, -37.059, 5.775, -33.924, -4.797]
  MoveL (T16773) to (106.29, 103.84, 18.1) mm, rotated rx 180 ry 0 rz -180 deg; joints [3.219, 70.848, -37.059, 5.775, -33.924, -4.797]
  Set speed (40.0 mm/s)
  Call Extruder 2.0
  MoveL (T16774) to (106.29, 103.84, 18.1) mm, rotated rx 180 ry 0 rz -180 deg; joints [3.219, 70.848, -37.059, 5.775, -33.924, -4.797]
  Set speed (50.0 mm/s)
  MoveL (T16775) to (106.29, 103.84, 18.1) mm, rotated rx 180 ry 0 rz -180 deg; joints [3.219, 70.848, -37.059, 5.775, -33.924, -4.797]
  Call Extruder 0.07441
  MoveL (T16776) to (103.84, 103.84, 18.1) mm, rotated rx 180 ry 0 rz -180 deg; joints [3.219, 70.848, -37.059, 5.775, -33.924, -4.797]
  Call Extruder 0.07644
  MoveL (T16777) to (105.62, 105.62, 18.1) mm, rotated rx 180 ry 0 rz -180 deg; joints [3.219, 70.848, -37.059, 5.775, -33.924, -4.797]
  Call Extruder 0.00165
  MoveL (T16778) to (105.62, 105.56, 18.1) mm, rotated rx 180 ry 0 rz -180 deg; joints [3.219, 70.848, -37.059, 5.775, -33.924, -4.797]
  Call Extruder 0.07644
  MoveL (T16779) to (103.84, 107.34, 18.1) mm, rotated rx 180 ry 0 rz -180 deg; joints [3.219, 70.615, -37.016, 5.804, -33.735, -4.832]
  Call Extruder 0.03385
  MoveL (T16780) to (103.84, 108.45, 18.1) mm, rotated rx 180 ry 0 rz -180 deg; joints [1.407, 66.075, -28.498, 2.307, -37.6, -1.828]
  Call Extruder 0.18981
  MoveL (T16781) to (108.25, 112.86, 18.1) mm, rotated rx 180 ry 0 rz -180 deg; joints [1.407, 66.288, -28.531, 2.298, -37.78, -1.816]
  Call Extruder 0.04262
  MoveL (T16782) to (108.89, 114.1, 18.1) mm, rotated rx 180 ry 0 rz -180 deg; joints [1.407, 66.288, -28.531, 2.298, -37.78, -1.816]
  Call Extruder 0.0398
  MoveL (T16783) to (107.58, 114.1, 18.1) mm, rotated rx 180 ry 0 rz -180 deg; joints [1.407, 66.288, -28.531, 2.298, -37.78, -1.816]
  Call Extruder 0.05791
  MoveL (T16784) to (106.23, 115.45, 18.1) mm, rotated rx 180 ry 0 rz -180 deg; joints [1.407, 66.288, -28.531, 2.298, -37.78, -1.816]
  Call Extruder 0.10299
  MoveL (T16785) to (103.84, 113.06, 18.1) mm, rotated rx 180 ry 0 rz -180 deg; joints [1.407, 66.288, -28.531, 2.298, -37.78, -1.816]
  Call Extruder 0.03385
  MoveL (T16786) to (103.84, 111.94, 18.1) mm, rotated rx 180 ry 0 rz -180 deg; joints [1.363, 71.129, -37.626, 2.469, -33.528, -2.058]
  Call Extruder 0.11243
  MoveL (T16787) to (106.45, 109.33, 18.1) mm, rotated rx 180 ry 0 rz -180 deg; joints [1.363, 71.129, -37.626, 2.469, -33.528, -2.058]
  Call Extruder 0.04411
  MoveL (T16788) to (105.8, 108.05, 18.1) mm, rotated rx 180 ry 0 rz -180 deg; joints [1.363, 71.129, -37.626, 2.469, -33.528, -2.058]
  Call Extruder 0.02313
  MoveL (T16789) to (105.62, 107.31, 18.1) mm, rotated rx 180 ry 0 rz -180 deg; joints [3.241, 71.356, -38.053, 5.889, -33.443, -4.919]
  Call Extruder 0.00717
  MoveL (T16790) to (105.62, 107.07, 18.1) mm, rotated rx 180 ry 0 rz -180 deg; joints [3.241, 71.356, -38.053, 5.889, -33.443, -4.919]
  Set speed (45.0 mm/s)
  Call Extruder -1.6
  MoveL (T16791) to (105.62, 107.07, 18.1) mm, rotated rx 180 ry 0 rz -180 deg; joints [3.351, 66.274, -28.504, 5.461, -37.896, -4.314]
  Set speed (120.0 mm/s)
  MoveL (T16792) to (105.62, 107.07, 18.1) mm, rotated rx 180 ry 0 rz -180 deg; joints [3.351, 66.274, -28.504, 5.461, -37.896, -4.314]
  Call Extruder -0.08383
  MoveL (T16793) to (105.62, 107.31, 18.1) mm, rotated rx 180 ry 0 rz -180 deg; joints [3.351, 66.274, -28.504, 5.461, -37.896, -4.314]
  Call Extruder -0.27043
  MoveL (T16794) to (105.8, 108.05, 18.1) mm, rotated rx 180 ry 0 rz -180 deg; joints [3.351, 66.274, -28.504, 5.461, -37.896, -4.314]
  Call Extruder -0.02574
  MoveL (T16795) to (105.83, 108.11, 18.1) mm, rotated rx 180 ry 0 rz -180 deg; joints [1.409, 66.083, -28.145, 2.292, -37.96, -1.807]
  Set speed (45.0 mm/s)
  Call Extruder -0.02
  MoveL (T16796) to (105.83, 108.11, 18.1) mm, rotated rx 180 ry 0 rz -180 deg; joints [1.409, 66.083, -28.145, 2.292, -37.96, -1.807]
  Set speed (150.0 mm/s)
  MoveL (T16797) to (105.83, 108.11, 20.1) mm, rotated rx 180 ry 0 rz -180 deg; joints [1.409, 66.083, -28.145, 2.292, -37.96, -1.807]
  MoveL (T16798) to (108.01, 112.39, 20.1) mm, rotated rx 180 ry 0 rz -180 deg; joints [1.407, 66.273, -28.502, 2.297, -37.793, -1.816]
  MoveL (T16799) to (108.01, 112.39, 18.1) mm, rotated rx 180 ry 0 rz -180 deg; joints [1.407, 66.273, -28.502, 2.297, -37.793, -1.816]
  Set speed (40.0 mm/s)
  Call Extruder 2.0
  MoveL (T16800) to (108.01, 112.39, 18.1) mm, rotated rx 180 ry 0 rz -180 deg; joints [1.365, 66.078, -28.137, 2.22, -37.962, -1.751]
  Set speed (50.0 mm/s)
  MoveL (T16801) to (108.01, 112.39, 18.1) mm, rotated rx 180 ry 0 rz -180 deg; joints [1.365, 66.078, -28.137, 2.22, -37.962, -1.751]
  Call Extruder 0.17945
  MoveL (T16802) to (103.84, 116.55, 18.1) mm, rotated rx 180 ry 0 rz -180 deg; joints [1.365, 66.078, -28.137, 2.22, -37.962, -1.751]
  Call Extruder 0.03385
  MoveL (T16803) to (103.84, 117.66, 18.1) mm, rotated rx 180 ry 0 rz -180 deg; joints [1.365, 66.078, -28.137, 2.22, -37.962, -1.751]
  Call Extruder 0.08006
  MoveL (T16804) to (105.7, 119.52, 18.1) mm, rotated rx 180 ry 0 rz -180 deg; joints [1.365, 66.078, -28.137, 2.22, -37.962, -1.751]
  Call Extruder 0.00677
  MoveL (T16805) to (105.7, 119.3, 18.1) mm, rotated rx 180 ry 0 rz -180 deg; joints [1.319, 71.254, -37.861, 2.396, -33.416, -2.001]
  Call Extruder 0.08006
  MoveL (T16806) to (103.84, 121.16, 18.1) mm, rotated rx 180 ry 0 rz -180 deg; joints [1.319, 71.254, -37.861, 2.396, -33.416, -2.001]
  Call Extruder 0.07441
  MoveL (T16807) to (106.29, 121.16, 18.1) mm, rotated rx 180 ry 0 rz -180 deg; joints [1.319, 71.254, -37.861, 2.396, -33.416, -2.001]
  Set speed (45.0 mm/s)
  Call Extruder -1.6
  MoveL (T16808) to (106.29, 121.16, 18.1) mm, rotated rx 180 ry 0 rz -180 deg; joints [3.282, 71.493, -38.31, 5.98, -33.327, -5.002]
  Set speed (120.0 mm/s)
  MoveL (T16809) to (106.29, 121.16, 18.1) mm, rotated rx 180 ry 0 rz -180 deg; joints [3.282, 71.493, -38.31, 5.98, -33.327, -5.002]
  Call Extruder -0.38
  MoveL (T16810) to (105.22, 121.16, 18.1) mm, rotated rx 180 ry 0 rz -180 deg; joints [3.398, 66.176, -28.32, 5.526, -37.985, -4.361]
  Set speed (45.0 mm/s)
  Call Extruder -0.02
  MoveL (T16811) to (105.22, 121.16, 18.1) mm, rotated rx 180 ry 0 rz -180 deg; joints [1.366, 65.976, -27.946, 2.217, -38.052, -1.746]
  Set speed (150.0 mm/s)
  MoveL (T16812) to (105.22, 121.16, 20.1) mm, rotated rx 180 ry 0 rz -180 deg; joints [1.366, 65.976, -27.946, 2.217, -38.052, -1.746]
  MoveL (T16813) to (118.71, 121.16, 20.1) mm, rotated rx 180 ry 0 rz -180 deg; joints [1.365, 66.063, -28.108, 2.219, -37.976, -1.75]
  MoveL (T16814) to (118.71, 121.16, 18.1) mm, rotated rx 180 ry 0 rz -180 deg; joints [1.365, 66.063, -28.108, 2.219, -37.976, -1.75]
  Set speed (40.0 mm/s)
  Call Extruder 2.0
  MoveL (T16815) to (118.71, 121.16, 18.1) mm, rotated rx 180 ry 0 rz -180 deg; joints [1.365, 66.063, -28.108, 2.219, -37.976, -1.75]
  Set speed (50.0 mm/s)
  MoveL (T16816) to (118.71, 121.16, 18.1) mm, rotated rx 180 ry 0 rz -180 deg; joints [1.365, 66.063, -28.108, 2.219, -37.976, -1.75]
  Call Extruder 0.07441
  MoveL (T16817) to (121.16, 121.16, 18.1) mm, rotated rx 180 ry 0 rz -180 deg; joints [1.332, 65.871, -27.748, 2.158, -38.143, -1.697]
  Call Extruder 0.06569
  MoveL (T16818) to (119.63, 119.63, 18.1) mm, rotated rx 180 ry 0 rz -180 deg; joints [1.332, 65.871, -27.748, 2.158, -38.143, -1.697]
  Call Extruder 0.01356
  MoveL (T16819) to (119.63, 119.19, 18.1) mm, rotated rx 180 ry 0 rz -180 deg; joints [1.332, 65.871, -27.748, 2.158, -38.143, -1.697]
  Call Extruder 0.06569
  MoveL (T16820) to (121.16, 117.66, 18.1) mm, rotated rx 180 ry 0 rz -180 deg; joints [1.323, 65.87, -27.747, 2.143, -38.143, -1.685]
  Call Extruder 0.03385
  MoveL (T16821) to (121.16, 116.55, 18.1) mm, rotated rx 180 ry 0 rz -180 deg; joints [1.323, 65.87, -27.747, 2.143, -38.143, -1.685]
  Call Extruder 0.18312
  MoveL (T16822) to (116.91, 112.3, 18.1) mm, rotated rx 180 ry 0 rz -180 deg; joints [1.276, 71.38, -38.097, 2.324, -33.304, -1.943]
  Call Extruder 0.00907
  MoveL (T16823) to (117.04, 112.56, 18.1) mm, rotated rx 180 ry 0 rz -180 deg; joints [1.276, 71.38, -38.097, 2.324, -33.304, -1.943]
  Call Extruder 0.17727
  MoveL (T16824) to (121.16, 108.45, 18.1) mm, rotated rx 180 ry 0 rz -180 deg; joints [3.322, 71.63, -38.568, 6.073, -33.21, -5.086]
  Call Extruder 0.03385
  MoveL (T16825) to (121.16, 107.34, 18.1) mm, rotated rx 180 ry 0 rz -180 deg; joints [3.322, 71.63, -38.568, 6.073, -33.21, -5.086]
  Call Extruder 0.05772
  MoveL (T16826) to (119.82, 106, 18.1) mm, rotated rx 180 ry 0 rz -180 deg; joints [3.445, 66.078, -28.136, 5.591, -38.075, -4.407]
  Call Extruder 0.02482
  MoveL (T16827) to (119.82, 105.18, 18.1) mm, rotated rx 180 ry 0 rz -180 deg; joints [3.445, 66.078, -28.136, 5.591, -38.075, -4.407]
  Call Extruder 0.05772
  MoveL (T16828) to (121.16, 103.84, 18.1) mm, rotated rx 180 ry 0 rz -180 deg; joints [1.339, 65.871, -27.748, 2.168, -38.143, -1.706]
  Call Extruder 0.07441
  MoveL (T16829) to (118.71, 103.84, 18.1) mm, rotated rx 180 ry 0 rz -180 deg; joints [1.339, 65.871, -27.748, 2.168, -38.143, -1.706]
  Set speed (45.0 mm/s)
  Call Extruder -1.6
  MoveL (T16830) to (118.71, 103.84, 18.1) mm, rotated rx 180 ry 0 rz -180 deg; joints [1.326, 65.886, -27.775, 2.147, -38.13, -1.69]
  Set speed (120.0 mm/s)
  MoveL (T16831) to (118.71, 103.84, 18.1) mm, rotated rx 180 ry 0 rz -180 deg; joints [1.326, 65.886, -27.775, 2.147, -38.13, -1.69]
  Call Extruder -0.38
  MoveL (T16832) to (119.78, 103.84, 18.1) mm, rotated rx 180 ry 0 rz -180 deg; joints [1.326, 65.886, -27.775, 2.147, -38.13, -1.69]
  Set speed (45.0 mm/s)
  Call Extruder -0.02
  MoveL (T16833) to (119.78, 103.84, 18.1) mm, rotated rx 180 ry 0 rz -180 deg; joints [1.326, 65.886, -27.775, 2.147, -38.13, -1.69]
  Set speed (150.0 mm/s)
  MoveL (T16834) to (119.78, 103.84, 20.1) mm, rotated rx 180 ry 0 rz -180 deg; joints [1.326, 65.886, -27.775, 2.147, -38.13, -1.69]
  MoveL (T16835) to (119.19, 109.98, 20.1) mm, rotated rx 180 ry 0 rz -180 deg; joints [1.326, 65.886, -27.775, 2.147, -38.13, -1.69]
  MoveL (T16836) to (119.19, 109.98, 18.1) mm, rotated rx 180 ry 0 rz -180 deg; joints [1.326, 65.886, -27.775, 2.147, -38.13, -1.69]
  Set speed (40.0 mm/s)
  Call Extruder 2.0
  MoveL (T16837) to (119.19, 109.98, 18.1) mm, rotated rx 180 ry 0 rz -180 deg; joints [1.326, 65.886, -27.775, 2.147, -38.13, -1.69]
  Set speed (50.0 mm/s)
  MoveL (T16838) to (119.19, 109.98, 18.1) mm, rotated rx 180 ry 0 rz -180 deg; joints [1.323, 65.87, -27.747, 2.143, -38.143, -1.685]
  Call Extruder 0.08482
  MoveL (T16839) to (121.16, 111.94, 18.1) mm, rotated rx 180 ry 0 rz -180 deg; joints [1.323, 65.87, -27.747, 2.143, -38.143, -1.685]
  Call Extruder 0.03385
  MoveL (T16840) to (121.16, 113.06, 18.1) mm, rotated rx 180 ry 0 rz -180 deg; joints [1.323, 65.87, -27.747, 2.143, -38.143, -1.685]
  Call Extruder 0.1101
  MoveL (T16841) to (118.6, 115.61, 18.1) mm, rotated rx 180 ry 0 rz -180 deg; joints [1.321, 66.105, -28.188, 2.149, -37.937, -1.695]
  Call Extruder 0.05702
  MoveL (T16842) to (119.45, 117.28, 18.1) mm, rotated rx 180 ry 0 rz -180 deg; joints [1.321, 66.105, -28.188, 2.149, -37.937, -1.695]
  Call Extruder 0.01739
  MoveL (T16843) to (119.59, 117.83, 18.1) mm, rotated rx 180 ry 0 rz -180 deg; joints [1.321, 66.105, -28.188, 2.149, -37.937, -1.695]
  Set speed (45.0 mm/s)
  Call Extruder -1.6
  MoveL (T16844) to (119.59, 117.83, 18.1) mm, rotated rx 180 ry 0 rz -180 deg; joints [1.321, 66.105, -28.188, 2.149, -37.937, -1.695]
  Set speed (120.0 mm/s)
  MoveL (T16845) to (119.59, 117.83, 18.1) mm, rotated rx 180 ry 0 rz -180 deg; joints [1.321, 66.105, -28.188, 2.149, -37.937, -1.695]
  Call Extruder -0.20338
  MoveL (T16846) to (119.45, 117.28, 18.1) mm, rotated rx 180 ry 0 rz -180 deg; joints [1.321, 66.105, -28.188, 2.149, -37.937, -1.695]
  Call Extruder -0.17662
  MoveL (T16847) to (119.23, 116.84, 18.1) mm, rotated rx 180 ry 0 rz -180 deg; joints [1.707, 66.18, -28.328, 2.78, -37.885, -2.194]
  Set speed (45.0 mm/s)
  Call Extruder -0.02
  MoveL (T16848) to (119.23, 116.84, 18.1) mm, rotated rx 180 ry 0 rz -180 deg; joints [1.707, 66.18, -28.328, 2.78, -37.885, -2.194]
  Set speed (150.0 mm/s)
  MoveL (T16849) to (119.23, 116.84, 20.1) mm, rotated rx 180 ry 0 rz -180 deg; joints [1.707, 66.18, -28.328, 2.78, -37.885, -2.194]
  MoveL (T16850) to (119.41, 119.83, 20.1) mm, rotated rx 180 ry 0 rz -180 deg; joints [1.707, 66.18, -28.328, 2.78, -37.885, -2.194]
  MoveL (T16851) to (119.41, 119.83, 18.1) mm, rotated rx 180 ry 0 rz -180 deg; joints [1.707, 66.18, -28.328, 2.78, -37.885, -2.194]
  Set speed (40.0 mm/s)
  Call Extruder 2.0
  MoveL (T16852) to (119.41, 119.83, 18.1) mm, rotated rx 180 ry 0 rz -180 deg; joints [1.707, 66.18, -28.328, 2.78, -37.885, -2.194]
  Set speed (25.0 mm/s)
  MoveL (T16853) to (119.41, 119.83, 18.1) mm, rotated rx 180 ry 0 rz -180 deg; joints [1.707, 66.18, -28.328, 2.78, -37.885, -2.194]
  Call Extruder 0.05145
  MoveL (T16854) to (118.05, 121.18, 18.1) mm, rotated rx 180 ry 0 rz -180 deg; joints [1.707, 66.18, -28.328, 2.78, -37.885, -2.194]
  Call Extruder 0.01361
  MoveL (T16855) to (117.55, 121.18, 18.1) mm, rotated rx 180 ry 0 rz -180 deg; joints [1.707, 66.18, -28.328, 2.78, -37.885, -2.194]
  Call Extruder 0.0646
  MoveL (T16856) to (119.25, 119.48, 18.1) mm, rotated rx 180 ry 0 rz -180 deg; joints [1.707, 66.18, -28.328, 2.78, -37.885, -2.194]
  Call Extruder 0.01361
  MoveL (T16857) to (119.25, 118.97, 18.1) mm, rotated rx 180 ry 0 rz -180 deg; joints [1.707, 66.18, -28.328, 2.78, -37.885, -2.194]
  Call Extruder 0.08385
  MoveL (T16858) to (117.04, 121.18, 18.1) mm, rotated rx 180 ry 0 rz -180 deg; joints [1.442, 66.163, -28.296, 2.348, -37.891, -1.853]
  Call Extruder 0.01361
  MoveL (T16859) to (116.53, 121.18, 18.1) mm, rotated rx 180 ry 0 rz -180 deg; joints [1.442, 66.163, -28.296, 2.348, -37.891, -1.853]
  Call Extruder 0.1031
  MoveL (T16860) to (119.25, 118.46, 18.1) mm, rotated rx 180 ry 0 rz -180 deg; joints [1.442, 66.163, -28.296, 2.348, -37.891, -1.853]
  Call Extruder 0.01077
  MoveL (T16861) to (119.25, 118.06, 18.1) mm, rotated rx 180 ry 0 rz -180 deg; joints [1.657, 66.178, -28.324, 2.699, -37.885, -2.131]
  Call Extruder 0.00235
  MoveL (T16862) to (119.23, 117.98, 18.1) mm, rotated rx 180 ry 0 rz -180 deg; joints [1.657, 66.178, -28.324, 2.699, -37.885, -2.131]
  Call Extruder 0.12157
  MoveL (T16863) to (116.03, 121.18, 18.1) mm, rotated rx 180 ry 0 rz -180 deg; joints [1.657, 66.178, -28.324, 2.699, -37.885, -2.131]
  Call Extruder 0.01361
  MoveL (T16864) to (115.52, 121.18, 18.1) mm, rotated rx 180 ry 0 rz -180 deg; joints [1.679, 66.201, -28.367, 2.736, -37.866, -2.16]
  Call Extruder 0.13708
  MoveL (T16865) to (119.13, 117.57, 18.1) mm, rotated rx 180 ry 0 rz -180 deg; joints [1.679, 66.201, -28.367, 2.736, -37.866, -2.16]
  Call Extruder 0.00436
  MoveL (T16866) to (119.09, 117.41, 18.1) mm, rotated rx 180 ry 0 rz -180 deg; joints [1.743, 66.362, -28.67, 2.849, -37.726, -2.254]
  Call Extruder 0.00621
  MoveL (T16867) to (118.99, 117.2, 18.1) mm, rotated rx 180 ry 0 rz -180 deg; joints [1.743, 66.362, -28.67, 2.849, -37.726, -2.254]
  Call Extruder 0.15089
  MoveL (T16868) to (115.01, 121.18, 18.1) mm, rotated rx 180 ry 0 rz -180 deg; joints [1.743, 66.362, -28.67, 2.849, -37.726, -2.254]
  Call Extruder 0.01361
  MoveL (T16869) to (114.5, 121.18, 18.1) mm, rotated rx 180 ry 0 rz -180 deg; joints [1.821, 66.188, -28.344, 2.966, -37.882, -2.342]
  Call Extruder 0.16362
  MoveL (T16870) to (118.81, 116.87, 18.1) mm, rotated rx 180 ry 0 rz -180 deg; joints [1.821, 66.188, -28.344, 2.966, -37.882, -2.342]
  Call Extruder 0.01011
  MoveL (T16871) to (118.64, 116.53, 18.1) mm, rotated rx 180 ry 0 rz -180 deg; joints [1.821, 66.188, -28.344, 2.966, -37.882, -2.342]
  Call Extruder 0.17635
  MoveL (T16872) to (114, 121.18, 18.1) mm, rotated rx 180 ry 0 rz -180 deg; joints [1.821, 66.188, -28.344, 2.966, -37.882, -2.342]
  Call Extruder 0.01361
  MoveL (T16873) to (113.49, 121.18, 18.1) mm, rotated rx 180 ry 0 rz -180 deg; joints [1.941, 66.198, -28.361, 3.162, -37.879, -2.497]
  Call Extruder 0.18908
  MoveL (T16874) to (118.47, 116.2, 18.1) mm, rotated rx 180 ry 0 rz -180 deg; joints [1.941, 66.198, -28.361, 3.162, -37.879, -2.497]
  Call Extruder 0.01011
  MoveL (T16875) to (118.3, 115.86, 18.1) mm, rotated rx 180 ry 0 rz -180 deg; joints [3.239, 69.848, -35.219, 5.686, -34.761, -4.676]
  Call Extruder 0.20182
  MoveL (T16876) to (112.98, 121.18, 18.1) mm, rotated rx 180 ry 0 rz -180 deg; joints [3.239, 69.848, -35.219, 5.686, -34.761, -4.676]
  Call Extruder 0.01361
  MoveL (T16877) to (112.47, 121.18, 18.1) mm, rotated rx 180 ry 0 rz -180 deg; joints [3.232, 70.18, -35.842, 5.717, -34.471, -4.718]
  Call Extruder 0.21455
  MoveL (T16878) to (118.13, 115.53, 18.1) mm, rotated rx 180 ry 0 rz -180 deg; joints [3.232, 70.18, -35.842, 5.717, -34.471, -4.718]
  Call Extruder 0.01011
  MoveL (T16879) to (117.96, 115.19, 18.1) mm, rotated rx 180 ry 0 rz -180 deg; joints [3.232, 70.18, -35.842, 5.717, -34.471, -4.718]
  Call Extruder 0.22728
  MoveL (T16880) to (111.97, 121.18, 18.1) mm, rotated rx 180 ry 0 rz -180 deg; joints [2.845, 71.196, -37.752, 5.153, -33.551, -4.298]
  Call Extruder 0.01361
  MoveL (T16881) to (111.46, 121.18, 18.1) mm, rotated rx 180 ry 0 rz -180 deg; joints [2.845, 71.196, -37.752, 5.153, -33.551, -4.298]
  Call Extruder 0.24002
  MoveL (T16882) to (117.78, 114.86, 18.1) mm, rotated rx 180 ry 0 rz -180 deg; joints [2.845, 71.196, -37.752, 5.153, -33.551, -4.298]
  Call Extruder 0.01011
  MoveL (T16883) to (117.61, 114.52, 18.1) mm, rotated rx 180 ry 0 rz -180 deg; joints [3.211, 71.254, -37.861, 5.821, -33.529, -4.857]
  Call Extruder 0.25275
  MoveL (T16884) to (110.95, 121.18, 18.1) mm, rotated rx 180 ry 0 rz -180 deg; joints [3.211, 71.254, -37.861, 5.821, -33.529, -4.857]
  Call Extruder 0.01361
  MoveL (T16885) to (110.45, 121.18, 18.1) mm, rotated rx 180 ry 0 rz -180 deg; joints [1.893, 67.324, -30.476, 3.155, -36.89, -2.524]
  Call Extruder 0.26548
  MoveL (T16886) to (117.44, 114.19, 18.1) mm, rotated rx 180 ry 0 rz -180 deg; joints [1.893, 67.324, -30.476, 3.155, -36.89, -2.524]
  Call Extruder 0.01011
  MoveL (T16887) to (117.27, 113.85, 18.1) mm, rotated rx 180 ry 0 rz -180 deg; joints [1.893, 67.324, -30.476, 3.155, -36.89, -2.524]
  Call Extruder 0.27822
  MoveL (T16888) to (109.94, 121.18, 18.1) mm, rotated rx 180 ry 0 rz -180 deg; joints [1.895, 67.187, -30.219, 3.149, -37.01, -2.515]
  Call Extruder 0.01361
  MoveL (T16889) to (109.43, 121.18, 18.1) mm, rotated rx 180 ry 0 rz -180 deg; joints [1.895, 67.187, -30.219, 3.149, -37.01, -2.515]
  Call Extruder 0.29095
  MoveL (T16890) to (117.1, 113.52, 18.1) mm, rotated rx 180 ry 0 rz -180 deg; joints [2.319, 66.231, -28.424, 3.78, -37.868, -2.986]
  Call Extruder 0.01011
  MoveL (T16891) to (116.93, 113.18, 18.1) mm, rotated rx 180 ry 0 rz -180 deg; joints [2.319, 66.231, -28.424, 3.78, -37.868, -2.986]
  Call Extruder 0.30368
  MoveL (T16892) to (108.92, 121.18, 18.1) mm, rotated rx 180 ry 0 rz -180 deg; joints [2.44, 66.243, -28.446, 3.977, -37.864, -3.142]
  Call Extruder 0.01361
  MoveL (T16893) to (108.42, 121.18, 18.1) mm, rotated rx 180 ry 0 rz -180 deg; joints [3.266, 68.523, -32.728, 5.573, -35.923, -4.518]
  Call Extruder 0.31641
  MoveL (T16894) to (116.75, 112.84, 18.1) mm, rotated rx 180 ry 0 rz -180 deg; joints [3.266, 68.523, -32.728, 5.573, -35.923, -4.518]
  Call Extruder 0.01011
  MoveL (T16895) to (116.58, 112.51, 18.1) mm, rotated rx 180 ry 0 rz -180 deg; joints [3.26, 68.836, -33.317, 5.599, -35.649, -4.554]
  Call Extruder 0.32915
  MoveL (T16896) to (107.91, 121.18, 18.1) mm, rotated rx 180 ry 0 rz -180 deg; joints [3.26, 68.836, -33.317, 5.599, -35.649, -4.554]
  Call Extruder 0.01361
  MoveL (T16897) to (107.4, 121.18, 18.1) mm, rotated rx 180 ry 0 rz -180 deg; joints [2.685, 70.268, -36.007, 4.761, -34.353, -3.934]
  Call Extruder 0.34188
  MoveL (T16898) to (116.41, 112.17, 18.1) mm, rotated rx 180 ry 0 rz -180 deg; joints [2.685, 70.268, -36.007, 4.761, -34.353, -3.934]
  Call Extruder 0.01011
  MoveL (T16899) to (116.24, 111.84, 18.1) mm, rotated rx 180 ry 0 rz -180 deg; joints [2.685, 70.268, -36.007, 4.761, -34.353, -3.934]
  Call Extruder 0.34736
  MoveL (T16900) to (107.09, 120.99, 18.1) mm, rotated rx 180 ry 0 rz -180 deg; joints [2.754, 70.487, -36.42, 4.908, -34.165, -4.064]
  Call Extruder 0.00962
  MoveL (T16901) to (106.83, 120.74, 18.1) mm, rotated rx 180 ry 0 rz -180 deg; joints [2.754, 70.487, -36.42, 4.908, -34.165, -4.064]
  Call Extruder 0.355
  MoveL (T16902) to (116.19, 111.38, 18.1) mm, rotated rx 180 ry 0 rz -180 deg; joints [2.754, 70.487, -36.42, 4.908, -34.165, -4.064]
  Set speed (150.0 mm/s)
  MoveL (T16903) to (117.58, 111, 18.1) mm, rotated rx 180 ry 0 rz -180 deg; joints [2.754, 70.487, -36.42, 4.908, -34.165, -4.064]
  Set speed (25.0 mm/s)
  MoveL (T16904) to (117.58, 111, 18.1) mm, rotated rx 180 ry 0 rz -180 deg; joints [2.762, 70.55, -36.537, 4.929, -34.111, -4.084]
  Call Extruder 0.07028
  MoveL (T16905) to (119.43, 109.15, 18.1) mm, rotated rx 180 ry 0 rz -180 deg; joints [2.756, 70.933, -37.258, 4.961, -33.774, -4.127]
  Call Extruder 0.01361
  MoveL (T16906) to (119.43, 108.64, 18.1) mm, rotated rx 180 ry 0 rz -180 deg; joints [2.756, 70.933, -37.258, 4.961, -33.774, -4.127]
  Call Extruder 0.08343
  MoveL (T16907) to (117.24, 110.84, 18.1) mm, rotated rx 180 ry 0 rz -180 deg; joints [2.756, 70.933, -37.258, 4.961, -33.774, -4.127]
  Call Extruder 0.01361
  MoveL (T16908) to (116.73, 110.84, 18.1) mm, rotated rx 180 ry 0 rz -180 deg; joints [2.756, 70.933, -37.258, 4.961, -33.774, -4.127]
  Call Extruder 0.10268
  MoveL (T16909) to (119.43, 108.14, 18.1) mm, rotated rx 180 ry 0 rz -180 deg; joints [2.731, 70.991, -37.367, 4.924, -33.722, -4.099]
  Call Extruder 0.01361
  MoveL (T16910) to (119.43, 107.63, 18.1) mm, rotated rx 180 ry 0 rz -180 deg; joints [2.731, 70.991, -37.367, 4.924, -33.722, -4.099]
  Call Extruder 0.12192
  MoveL (T16911) to (116.22, 110.84, 18.1) mm, rotated rx 180 ry 0 rz -180 deg; joints [2.731, 70.991, -37.367, 4.924, -33.722, -4.099]
  Call Extruder 0.01319
  MoveL (T16912) to (115.73, 110.84, 18.1) mm, rotated rx 180 ry 0 rz -180 deg; joints [2.731, 70.991, -37.367, 4.924, -33.722, -4.099]
  Call Extruder 0.0098
  MoveL (T16913) to (115.9, 111.17, 18.1) mm, rotated rx 180 ry 0 rz -180 deg; joints [2.662, 71.179, -37.72, 4.821, -33.552, -4.02]
  Call Extruder 0.35357
  MoveL (T16914) to (106.58, 120.48, 18.1) mm, rotated rx 180 ry 0 rz -180 deg; joints [2.662, 71.179, -37.72, 4.821, -33.552, -4.02]
  Call Extruder 0.00962
  MoveL (T16915) to (106.33, 120.23, 18.1) mm, rotated rx 180 ry 0 rz -180 deg; joints [2.61, 71.172, -37.707, 4.725, -33.555, -3.941]
  Call Extruder 0.49747
  MoveL (T16916) to (119.43, 107.12, 18.1) mm, rotated rx 180 ry 0 rz -180 deg; joints [2.61, 71.172, -37.707, 4.725, -33.555, -3.941]
  Call Extruder 0.01361
  MoveL (T16917) to (119.43, 106.61, 18.1) mm, rotated rx 180 ry 0 rz -180 deg; joints [2.61, 71.172, -37.707, 4.725, -33.555, -3.941]
  Call Extruder 0.50664
  MoveL (T16918) to (106.08, 119.96, 18.1) mm, rotated rx 180 ry 0 rz -180 deg; joints [2.717, 70.882, -37.162, 4.886, -33.817, -4.062]
  Call Extruder 0.01361
  MoveL (T16919) to (106.08, 119.46, 18.1) mm, rotated rx 180 ry 0 rz -180 deg; joints [2.717, 70.882, -37.162, 4.886, -33.817, -4.062]
  Call Extruder 0.50664
  MoveL (T16920) to (119.43, 106.11, 18.1) mm, rotated rx 180 ry 0 rz -180 deg; joints [2.719, 70.728, -36.871, 4.873, -33.952, -4.045]
  Call Extruder 0.01361
  MoveL (T16921) to (119.43, 105.6, 18.1) mm, rotated rx 180 ry 0 rz -180 deg; joints [2.719, 70.728, -36.871, 4.873, -33.952, -4.045]
  Call Extruder 0.50664
  MoveL (T16922) to (106.08, 118.95, 18.1) mm, rotated rx 180 ry 0 rz -180 deg; joints [2.557, 71.165, -37.693, 4.63, -33.558, -3.861]
  Call Extruder 0.01361
  MoveL (T16923) to (106.08, 118.44, 18.1) mm, rotated rx 180 ry 0 rz -180 deg; joints [2.557, 71.165, -37.693, 4.63, -33.558, -3.861]
  Call Extruder 0.50198
  MoveL (T16924) to (119.31, 105.22, 18.1) mm, rotated rx 180 ry 0 rz -180 deg; joints [2.505, 71.158, -37.68, 4.535, -33.56, -3.781]
  Call Extruder 0.00962
  MoveL (T16925) to (119.06, 104.96, 18.1) mm, rotated rx 180 ry 0 rz -180 deg; joints [2.505, 71.158, -37.68, 4.535, -33.56, -3.781]
  Call Extruder 0.49236
  MoveL (T16926) to (106.08, 117.94, 18.1) mm, rotated rx 180 ry 0 rz -180 deg; joints [2.722, 70.574, -36.583, 4.86, -34.087, -4.028]
  Call Extruder 0.01361
  MoveL (T16927) to (106.08, 117.43, 18.1) mm, rotated rx 180 ry 0 rz -180 deg; joints [2.722, 70.574, -36.583, 4.86, -34.087, -4.028]
  Call Extruder 0.11171
  MoveL (T16928) to (109.03, 114.48, 18.1) mm, rotated rx 180 ry 0 rz -180 deg; joints [2.722, 70.574, -36.583, 4.86, -34.087, -4.028]
  Call Extruder 0.01292
  MoveL (T16929) to (109.51, 114.48, 18.1) mm, rotated rx 180 ry 0 rz -180 deg; joints [2.719, 70.548, -36.534, 4.853, -34.11, -4.021]
  Call Extruder 0.00961
  MoveL (T16930) to (109.35, 114.17, 18.1) mm, rotated rx 180 ry 0 rz -180 deg; joints [2.719, 70.548, -36.534, 4.853, -34.11, -4.021]
  Call Extruder 0.35892
  MoveL (T16931) to (118.8, 104.71, 18.1) mm, rotated rx 180 ry 0 rz -180 deg; joints [2.719, 70.548, -36.534, 4.853, -34.11, -4.021]
  Call Extruder 0.00962
  MoveL (T16932) to (118.55, 104.45, 18.1) mm, rotated rx 180 ry 0 rz -180 deg; joints [2.719, 70.548, -36.534, 4.853, -34.11, -4.021]
  Call Extruder 0.3558
  MoveL (T16933) to (109.18, 113.83, 18.1) mm, rotated rx 180 ry 0 rz -180 deg; joints [2.7, 70.486, -36.417, 4.812, -34.163, -3.985]
  Call Extruder 0.01012
  MoveL (T16934) to (109, 113.49, 18.1) mm, rotated rx 180 ry 0 rz -180 deg; joints [2.453, 71.151, -37.668, 4.439, -33.563, -3.701]
  Call Extruder 0.35267
  MoveL (T16935) to (118.3, 104.2, 18.1) mm, rotated rx 180 ry 0 rz -180 deg; joints [2.453, 71.151, -37.668, 4.439, -33.563, -3.701]
  Call Extruder 0.00962
  MoveL (T16936) to (118.04, 103.95, 18.1) mm, rotated rx 180 ry 0 rz -180 deg; joints [2.4, 71.144, -37.655, 4.344, -33.565, -3.622]
  Call Extruder 0.34955
  MoveL (T16937) to (108.83, 113.16, 18.1) mm, rotated rx 180 ry 0 rz -180 deg; joints [2.4, 71.144, -37.655, 4.344, -33.565, -3.622]
  Call Extruder 0.01012
  MoveL (T16938) to (108.66, 112.82, 18.1) mm, rotated rx 180 ry 0 rz -180 deg; joints [2.675, 70.406, -36.268, 4.759, -34.231, -3.937]
  Call Extruder 0.34167
  MoveL (T16939) to (117.66, 103.82, 18.1) mm, rotated rx 180 ry 0 rz -180 deg; joints [2.675, 70.406, -36.268, 4.759, -34.231, -3.937]
  Call Extruder 0.01361
  MoveL (T16940) to (117.16, 103.82, 18.1) mm, rotated rx 180 ry 0 rz -180 deg; joints [2.65, 70.327, -36.119, 4.706, -34.298, -3.891]
  Call Extruder 0.32893
  MoveL (T16941) to (108.49, 112.49, 18.1) mm, rotated rx 180 ry 0 rz -180 deg; joints [2.65, 70.327, -36.119, 4.706, -34.298, -3.891]
  Call Extruder 0.01012
  MoveL (T16942) to (108.32, 112.15, 18.1) mm, rotated rx 180 ry 0 rz -180 deg; joints [2.65, 70.327, -36.119, 4.706, -34.298, -3.891]
  Call Extruder 0.31618
  MoveL (T16943) to (116.65, 103.82, 18.1) mm, rotated rx 180 ry 0 rz -180 deg; joints [2.348, 71.138, -37.643, 4.249, -33.568, -3.542]
  Call Extruder 0.01361
  MoveL (T16944) to (116.14, 103.82, 18.1) mm, rotated rx 180 ry 0 rz -180 deg; joints [2.348, 71.138, -37.643, 4.249, -33.568, -3.542]
  Call Extruder 0.30343
  MoveL (T16945) to (108.15, 111.81, 18.1) mm, rotated rx 180 ry 0 rz -180 deg; joints [2.348, 71.138, -37.643, 4.249, -33.568, -3.542]
  Call Extruder 0.01012
  MoveL (T16946) to (107.98, 111.48, 18.1) mm, rotated rx 180 ry 0 rz -180 deg; joints [2.295, 71.132, -37.631, 4.153, -33.57, -3.462]
  Call Extruder 0.29069
  MoveL (T16947) to (115.64, 103.82, 18.1) mm, rotated rx 180 ry 0 rz -180 deg; joints [2.295, 71.132, -37.631, 4.153, -33.57, -3.462]
  Call Extruder 0.01361
  MoveL (T16948) to (115.13, 103.82, 18.1) mm, rotated rx 180 ry 0 rz -180 deg; joints [2.295, 71.132, -37.631, 4.153, -33.57, -3.462]
  Call Extruder 0.27794
  MoveL (T16949) to (107.81, 111.14, 18.1) mm, rotated rx 180 ry 0 rz -180 deg; joints [2.295, 71.132, -37.631, 4.153, -33.57, -3.462]
  Call Extruder 0.01012
  MoveL (T16950) to (107.63, 110.81, 18.1) mm, rotated rx 180 ry 0 rz -180 deg; joints [2.625, 70.248, -35.97, 4.653, -34.366, -3.844]
  Call Extruder 0.26519
  MoveL (T16951) to (114.62, 103.82, 18.1) mm, rotated rx 180 ry 0 rz -180 deg; joints [2.625, 70.248, -35.97, 4.653, -34.366, -3.844]
  Call Extruder 0.01361
  MoveL (T16952) to (114.11, 103.82, 18.1) mm, rotated rx 180 ry 0 rz -180 deg; joints [2.625, 70.248, -35.97, 4.653, -34.366, -3.844]
  Call Extruder 0.25245
  MoveL (T16953) to (107.46, 110.47, 18.1) mm, rotated rx 180 ry 0 rz -180 deg; joints [2.625, 70.248, -35.97, 4.653, -34.366, -3.844]
  Call Extruder 0.01012
  MoveL (T16954) to (107.29, 110.14, 18.1) mm, rotated rx 180 ry 0 rz -180 deg; joints [2.599, 70.17, -35.823, 4.601, -34.433, -3.797]
  Call Extruder 0.2397
  MoveL (T16955) to (113.61, 103.82, 18.1) mm, rotated rx 180 ry 0 rz -180 deg; joints [2.599, 70.17, -35.823, 4.601, -34.433, -3.797]
  Call Extruder 0.01361
  MoveL (T16956) to (113.1, 103.82, 18.1) mm, rotated rx 180 ry 0 rz -180 deg; joints [2.599, 70.17, -35.823, 4.601, -34.433, -3.797]
  Call Extruder 0.22695
  MoveL (T16957) to (107.12, 109.8, 18.1) mm, rotated rx 180 ry 0 rz -180 deg; joints [2.243, 71.125, -37.619, 4.058, -33.572, -3.383]
  Call Extruder 0.01012
  MoveL (T16958) to (106.95, 109.46, 18.1) mm, rotated rx 180 ry 0 rz -180 deg; joints [2.243, 71.125, -37.619, 4.058, -33.572, -3.383]
  Call Extruder 0.21421
  MoveL (T16959) to (112.59, 103.82, 18.1) mm, rotated rx 180 ry 0 rz -180 deg; joints [2.243, 71.125, -37.619, 4.058, -33.572, -3.383]
  Call Extruder 0.01361
  MoveL (T16960) to (112.08, 103.82, 18.1) mm, rotated rx 180 ry 0 rz -180 deg; joints [2.19, 71.119, -37.608, 3.963, -33.575, -3.303]
  Call Extruder 0.20146
  MoveL (T16961) to (106.78, 109.13, 18.1) mm, rotated rx 180 ry 0 rz -180 deg; joints [2.19, 71.119, -37.608, 3.963, -33.575, -3.303]
  Call Extruder 0.01012
  MoveL (T16962) to (106.61, 108.79, 18.1) mm, rotated rx 180 ry 0 rz -180 deg; joints [2.19, 71.119, -37.608, 3.963, -33.575, -3.303]
  Call Extruder 0.18871
  MoveL (T16963) to (111.58, 103.82, 18.1) mm, rotated rx 180 ry 0 rz -180 deg; joints [2.19, 71.119, -37.608, 3.963, -33.575, -3.303]
  Call Extruder 0.01361
  MoveL (T16964) to (111.07, 103.82, 18.1) mm, rotated rx 180 ry 0 rz -180 deg; joints [2.574, 70.091, -35.675, 4.548, -34.5, -3.751]
  Call Extruder 0.17597
  MoveL (T16965) to (106.44, 108.46, 18.1) mm, rotated rx 180 ry 0 rz -180 deg; joints [2.574, 70.091, -35.675, 4.548, -34.5, -3.751]
  Call Extruder 0.01012
  MoveL (T16966) to (106.26, 108.12, 18.1) mm, rotated rx 180 ry 0 rz -180 deg; joints [2.574, 70.091, -35.675, 4.548, -34.5, -3.751]
  Call Extruder 0.16322
  MoveL (T16967) to (110.56, 103.82, 18.1) mm, rotated rx 180 ry 0 rz -180 deg; joints [2.549, 70.013, -35.529, 4.496, -34.567, -3.705]
  Call Extruder 0.01361
  MoveL (T16968) to (110.06, 103.82, 18.1) mm, rotated rx 180 ry 0 rz -180 deg; joints [2.549, 70.013, -35.529, 4.496, -34.567, -3.705]
  Call Extruder 0.14942
  MoveL (T16969) to (106.12, 107.76, 18.1) mm, rotated rx 180 ry 0 rz -180 deg; joints [2.549, 70.013, -35.529, 4.496, -34.567, -3.705]
  Call Extruder 0.01129
